LIN {X 0,Y 320.721,Z 461.024,A -85,B 0,C 180,E1 14265.571,E2 14265.571} C_VEL
LIN {X 0,Y 324.146,Z 440.908,A -85,B 0,C 180,E1 14264.497,E2 14264.497} C_VEL
LIN {X 0,Y 326.822,Z 419.622,A -85,B 0,C 180,E1 14263.687,E2 14263.687} C_VEL
LIN {X 0,Y 328.726,Z 391.924,A -85,B 0,C 180,E1 14262.985,E2 14262.985} C_VEL
LIN {X 0,Y 338,Z 225.821,A -85,B 0,C 180,E1 14259.275,E2 14259.275} C_VEL
LIN {X 0,Y 329.045,Z 209.572,A -85,B 0,C 180,E1 14256.958,E2 14256.958} C_VEL
LIN {X 0,Y 319.904,Z 194.705,A -85,B 0,C 180,E1 14254.397,E2 14254.397} C_VEL
LIN {X 0,Y 311.751,Z 182.649,A -85,B 0,C 180,E1 14251.896,E2 14251.896} C_VEL
LIN {X 0,Y 304.402,Z 172.591,A -85,B 0,C 180,E1 14249.41,E2 14249.41} C_VEL
LIN {X 0,Y 300.146,Z 166.89,A -85,B 0,C 180,E1 14247.799,E2 14247.799} C_VEL
LIN {X 0,Y 298.243,Z 163.151,A -85,B 0,C 180,E1 14246.265,E2 14246.265} C_VEL
LIN {X 0,Y 296.215,Z 159.192,A -85,B 0,C 180,E1 14244.53,E2 14244.53} C_VEL
LIN {X 0,Y 293.902,Z 154.755,A -85,B 0,C 180,E1 14242.397,E2 14242.397} C_VEL
LIN {X 0,Y 291.414,Z 150.066,A -85,B 0,C 180,E1 14239.857,E2 14239.857} C_VEL
LIN {X 0,Y 289.224,Z 146.434,A -85,B 0,C 180,E1 14237.503,E2 14237.503} C_VEL
LIN {X 0,Y 288.678,Z 145.099,A -85,B 0,C 180,E1 14236.707,E2 14236.707} C_VEL
LIN {X 0,Y 286.248,Z 141.602,A -85,B 0,C 180,E1 14233.74,E2 14233.74} C_VEL
LIN {X 0,Y 285.546,Z 139.698,A -85,B 0,C 180,E1 14232.333,E2 14232.333} C_VEL
LIN {X 0,Y 282.546,Z 135.185,A -85,B 0,C 180,E1 14226.706,E2 14226.706} C_VEL
LIN {X 0,Y 282.361,Z 134.287,A -85,B 0,C 180,E1 14225.282,E2 14225.282} C_VEL
LIN {X 0,Y 282.385,Z 134.265,A -85,B 0,C 180,E1 14220.608,E2 14220.608} C_VEL
LIN {X 0,Y 282.364,Z 134.277,A -85,B 0,C 180,E1 14215.938,E2 14215.938} C_VEL
LIN {X 0,Y 282.367,Z 134.308,A -85,B 0,C 180,E1 14211.08,E2 14211.08} C_VEL
LIN {X 0,Y 282.386,Z 134.493,A -85,B 0,C 180,E1 14209.596,E2 14209.596} C_VEL
LIN {X 0,Y 285.488,Z 139.677,A -85,B 0,C 180,E1 14203.1,E2 14203.1} C_VEL
LIN {X 0,Y 287.933,Z 144.473,A -85,B 0,C 180,E1 14199.255,E2 14199.255} C_VEL
LIN {X 0,Y 288.686,Z 145.379,A -85,B 0,C 180,E1 14198.461,E2 14198.461} C_VEL
LIN {X 0,Y 290.754,Z 149.516,A -85,B 0,C 180,E1 14195.843,E2 14195.843} C_VEL
LIN {X 0,Y 291.496,Z 150.817,A -85,B 0,C 180,E1 14195.045,E2 14195.045} C_VEL
LIN {X 0,Y 293.977,Z 155.554,A -85,B 0,C 180,E1 14192.447,E2 14192.447} C_VEL
LIN {X 0,Y 296.448,Z 160.545,A -85,B 0,C 180,E1 14190.054,E2 14190.054} C_VEL
LIN {X 0,Y 298.913,Z 165.761,A -85,B 0,C 180,E1 14187.807,E2 14187.807} C_VEL
LIN {X 0,Y 301.789,Z 171.506,A -85,B 0,C 180,E1 14185.605,E2 14185.605} C_VEL
LIN {X 0,Y 311.109,Z 184.598,A -85,B 0,C 180,E1 14182.393,E2 14182.393} C_VEL
LIN {X 0,Y 320.388,Z 199.042,A -85,B 0,C 180,E1 14179.556,E2 14179.556} C_VEL
LIN {X 0,Y 328.765,Z 213.325,A -85,B 0,C 180,E1 14177.237,E2 14177.237} C_VEL
LIN {X 0,Y 336.573,Z 228.034,A -85,B 0,C 180,E1 14175.231,E2 14175.231} C_VEL
LIN {X 0,Y 328.531,Z 396.994,A -85,B 0,C 180,E1 14171.76,E2 14171.76} C_VEL
LIN {X 0,Y 326.621,Z 416.539,A -85,B 0,C 180,E1 14171.071,E2 14171.071} C_VEL
LIN {X 0,Y 323.946,Z 435.192,A -85,B 0,C 180,E1 14170.112,E2 14170.112} C_VEL
LIN {X 0,Y 320.478,Z 453.585,A -85,B 0,C 180,E1 14168.835,E2 14168.835} C_VEL
LIN {X 0,Y 316.353,Z 471.266,A -85,B 0,C 180,E1 14167.245,E2 14167.245} C_VEL
LIN {X 0,Y 311.828,Z 487.803,A -85,B 0,C 180,E1 14165.362,E2 14165.362} C_VEL
LIN {X 0,Y 307.028,Z 503.233,A -85,B 0,C 180,E1 14163.167,E2 14163.167} C_VEL
LIN {X 0,Y 302.064,Z 517.674,A -85,B 0,C 180,E1 14160.612,E2 14160.612} C_VEL
LIN {X 0,Y 297.429,Z 530.269,A -85,B 0,C 180,E1 14157.856,E2 14157.856} C_VEL
LIN {X 0,Y 293.106,Z 541.516,A -85,B 0,C 180,E1 14154.807,E2 14154.807} C_VEL
LIN {X 0,Y 289.281,Z 551.303,A -85,B 0,C 180,E1 14151.491,E2 14151.491} C_VEL
LIN {X 0,Y 286.105,Z 559.611,A -85,B 0,C 180,E1 14147.909,E2 14147.909} C_VEL
LIN {X 0,Y 283.655,Z 566.396,A -85,B 0,C 180,E1 14144.075,E2 14144.075} C_VEL
LIN {X 0,Y 281.992,Z 571.558,A -85,B 0,C 180,E1 14140.004,E2 14140.004} C_VEL
LIN {X 0,Y 281.088,Z 574.878,A -85,B 0,C 180,E1 14135.92,E2 14135.92} C_VEL
LIN {X 0,Y 280.737,Z 576.48,A -85,B 0,C 180,E1 14131.836,E2 14131.836} C_VEL
LIN {X 0,Y 280.743,Z 576.471,A -85,B 0,C 180,E1 14127.958,E2 14127.958} C_VEL
LIN {X 0,Y 281.107,Z 574.834,A -85,B 0,C 180,E1 14123.873,E2 14123.873} C_VEL
LIN {X 0,Y 282.033,Z 571.47,A -85,B 0,C 180,E1 14119.789,E2 14119.789} C_VEL
LIN {X 0,Y 283.72,Z 566.25,A -85,B 0,C 180,E1 14115.717,E2 14115.717} C_VEL
LIN {X 0,Y 286.247,Z 559.287,A -85,B 0,C 180,E1 14111.824,E2 14111.824} C_VEL
LIN {X 0,Y 289.412,Z 551.061,A -85,B 0,C 180,E1 14108.304,E2 14108.304} C_VEL
LIN {X 0,Y 293.265,Z 541.222,A -85,B 0,C 180,E1 14104.989,E2 14104.989} C_VEL
LIN {X 0,Y 297.622,Z 529.918,A -85,B 0,C 180,E1 14101.943,E2 14101.943} C_VEL
LIN {X 0,Y 302.334,Z 517.118,A -85,B 0,C 180,E1 14099.161,E2 14099.161} C_VEL
LIN {X 0,Y 307.275,Z 502.717,A -85,B 0,C 180,E1 14096.637,E2 14096.637} C_VEL
LIN {X 0,Y 311.997,Z 487.513,A -85,B 0,C 180,E1 14094.489,E2 14094.489} C_VEL
LIN {X 0,Y 316.644,Z 470.484,A -85,B 0,C 180,E1 14092.564,E2 14092.564} C_VEL
LIN {X 0,Y 320.779,Z 452.575,A -85,B 0,C 180,E1 14090.976,E2 14090.976} C_VEL
LIN {X 0,Y 324.146,Z 434.561,A -85,B 0,C 180,E1 14089.741,E2 14089.741} C_VEL
LIN {X 0,Y 326.883,Z 415.161,A -85,B 0,C 180,E1 14088.763,E2 14088.763} C_VEL
LIN {X 0,Y 328.72,Z 395.639,A -85,B 0,C 180,E1 14088.095,E2 14088.095} C_VEL
LIN {X 0,Y 328.948,Z 391.546,A -85,B 0,C 180,E1 14087.996,E2 14087.996} C_VEL
LIN {X 0,Y 328.662,Z 383.97,A -85,B 0,C 180,E1 14087.703,E2 14087.703} C_VEL
LIN {X 0,Y 325.178,Z 364.134,A -85,B 0,C 180,E1 14086.515,E2 14086.515} C_VEL
LIN {X 0,Y 324.95,Z 357.606,A -85,B 0,C 180,E1 14086.286,E2 14086.286} C_VEL
LIN {X 0,Y 331.098,Z 230.961,A -85,B 0,C 180,E1 14083.663,E2 14083.663} C_VEL
LIN {X 0,Y 327.126,Z 223.644,A -85,B 0,C 180,E1 14082.619,E2 14082.619} C_VEL
LIN {X 0,Y 322.19,Z 240.736,A -85,B 0,C 180,E1 14082.119,E2 14082.119} C_VEL
LIN {X 0,Y 318.657,Z 249.667,A -85,B 0,C 180,E1 14081.638,E2 14081.638} C_VEL
LIN {X 0,Y 315.945,Z 253.882,A -85,B 0,C 180,E1 14081.167,E2 14081.167} C_VEL
LIN {X 0,Y 310.096,Z 277.776,A -85,B 0,C 180,E1 14080.634,E2 14080.634} C_VEL
LIN {X 0,Y 305.852,Z 291.273,A -85,B 0,C 180,E1 14080.092,E2 14080.092} C_VEL
LIN {X 0,Y 303.317,Z 296.772,A -85,B 0,C 180,E1 14079.663,E2 14079.663} C_VEL
LIN {X 0,Y 302.255,Z 297.734,A -85,B 0,C 180,E1 14079.431,E2 14079.431} C_VEL
LIN {X 0,Y 301.562,Z 297.398,A -85,B 0,C 180,E1 14079.232,E2 14079.232} C_VEL
LIN {X 0,Y 294.369,Z 406.379,A -85,B 0,C 180,E1 14075.561,E2 14075.561} C_VEL
LIN {X 0,Y 292.736,Z 426.04,A -85,B 0,C 180,E1 14074.541,E2 14074.541} C_VEL
LIN {X 0,Y 290.634,Z 445.674,A -85,B 0,C 180,E1 14073.162,E2 14073.162} C_VEL
LIN {X 0,Y 288.148,Z 465.179,A -85,B 0,C 180,E1 14071.392,E2 14071.392} C_VEL
LIN {X 0,Y 285.509,Z 483.447,A -85,B 0,C 180,E1 14069.306,E2 14069.306} C_VEL
LIN {X 0,Y 282.826,Z 500.339,A -85,B 0,C 180,E1 14066.905,E2 14066.905} C_VEL
LIN {X 0,Y 280.181,Z 516.365,A -85,B 0,C 180,E1 14064.118,E2 14064.118} C_VEL
LIN {X 0,Y 277.986,Z 529.646,A -85,B 0,C 180,E1 14061.302,E2 14061.302} C_VEL
LIN {X 0,Y 276.057,Z 541.908,A -85,B 0,C 180,E1 14058.149,E2 14058.149} C_VEL
LIN {X 0,Y 274.546,Z 552.542,A -85,B 0,C 180,E1 14054.77,E2 14054.77} C_VEL
LIN {X 0,Y 273.541,Z 561.1,A -85,B 0,C 180,E1 14051.384,E2 14051.384} C_VEL
LIN {X 0,Y 272.959,Z 567.848,A -85,B 0,C 180,E1 14048.002,E2 14048.002} C_VEL
LIN {X 0,Y 272.693,Z 573.226,A -85,B 0,C 180,E1 14044.417,E2 14044.417} C_VEL
LIN {X 0,Y 272.715,Z 576.877,A -85,B 0,C 180,E1 14040.841,E2 14040.841} C_VEL
LIN {X 0,Y 272.972,Z 578.945,A -85,B 0,C 180,E1 14037.271,E2 14037.271} C_VEL
LIN {X 0,Y 273.575,Z 579.472,A -85,B 0,C 180,E1 14033.706,E2 14033.706} C_VEL
LIN {X 0,Y 274.739,Z 578.347,A -85,B 0,C 180,E1 14029.94,E2 14029.94} C_VEL
LIN {X 0,Y 276.715,Z 575.316,A -85,B 0,C 180,E1 14025.99,E2 14025.99} C_VEL
LIN {X 0,Y 279.429,Z 570.626,A -85,B 0,C 180,E1 14022.293,E2 14022.293} C_VEL
LIN {X 0,Y 283.051,Z 564.115,A -85,B 0,C 180,E1 14018.664,E2 14018.664} C_VEL
LIN {X 0,Y 287.63,Z 555.651,A -85,B 0,C 180,E1 14015.127,E2 14015.127} C_VEL
LIN {X 0,Y 293.172,Z 544.938,A -85,B 0,C 180,E1 14011.702,E2 14011.702} C_VEL
LIN {X 0,Y 299.352,Z 532.673,A -85,B 0,C 180,E1 14008.598,E2 14008.598} C_VEL
LIN {X 0,Y 306.045,Z 518.945,A -85,B 0,C 180,E1 14005.811,E2 14005.811} C_VEL
LIN {X 0,Y 313.592,Z 502.655,A -85,B 0,C 180,E1 14003.172,E2 14003.172} C_VEL
LIN {X 0,Y 321.286,Z 485.354,A -85,B 0,C 180,E1 14000.936,E2 14000.936} C_VEL
LIN {X 0,Y 329.179,Z 466.218,A -85,B 0,C 180,E1 13998.999,E2 13998.999} C_VEL
LIN {X 0,Y 334.923,Z 451.016,A -85,B 0,C 180,E1 13997.764,E2 13997.764} C_VEL
LIN {X 0,Y 327.883,Z 467.006,A -85,B 0,C 180,E1 13996.661,E2 13996.661} C_VEL
LIN {X 0,Y 317.774,Z 488.595,A -85,B 0,C 180,E1 13994.688,E2 13994.688} C_VEL
LIN {X 0,Y 307.136,Z 511.532,A -85,B 0,C 180,E1 13991.865,E2 13991.865} C_VEL
LIN {X 0,Y 299.2,Z 529.521,A -85,B 0,C 180,E1 13989.046,E2 13989.046} C_VEL
LIN {X 0,Y 292.408,Z 545.751,A -85,B 0,C 180,E1 13986.026,E2 13986.026} C_VEL
LIN {X 0,Y 284.196,Z 568.647,A -85,B 0,C 180,E1 13980.859,E2 13980.859} C_VEL
LIN {X 0,Y 280.048,Z 581.452,A -85,B 0,C 180,E1 13977.252,E2 13977.252} C_VEL
LIN {X 0,Y 276.758,Z 592.506,A -85,B 0,C 180,E1 13973.417,E2 13973.417} C_VEL
LIN {X 0,Y 274.48,Z 601.426,A -85,B 0,C 180,E1 13969.582,E2 13969.582} C_VEL
LIN {X 0,Y 273.025,Z 608.934,A -85,B 0,C 180,E1 13965.507,E2 13965.507} C_VEL
LIN {X 0,Y 272.375,Z 614.641,A -85,B 0,C 180,E1 13961.435,E2 13961.435} C_VEL
LIN {X 0,Y 272.292,Z 618.543,A -85,B 0,C 180,E1 13957.385,E2 13957.385} C_VEL
LIN {X 0,Y 272.44,Z 620.7,A -85,B 0,C 180,E1 13953.578,E2 13953.578} C_VEL
LIN {X 0,Y 272.538,Z 621.429,A -85,B 0,C 180,E1 13950.001,E2 13950.001} C_VEL
LIN {X 0,Y 272.44,Z 620.694,A -85,B 0,C 180,E1 13946.424,E2 13946.424} C_VEL
LIN {X 0,Y 272.293,Z 618.427,A -85,B 0,C 180,E1 13942.494,E2 13942.494} C_VEL
LIN {X 0,Y 272.379,Z 614.605,A -85,B 0,C 180,E1 13938.553,E2 13938.553} C_VEL
LIN {X 0,Y 273.08,Z 608.583,A -85,B 0,C 180,E1 13934.281,E2 13934.281} C_VEL
LIN {X 0,Y 274.579,Z 600.957,A -85,B 0,C 180,E1 13930.207,E2 13930.207} C_VEL
LIN {X 0,Y 276.908,Z 591.911,A -85,B 0,C 180,E1 13926.373,E2 13926.373} C_VEL
LIN {X 0,Y 280.199,Z 580.888,A -85,B 0,C 180,E1 13922.594,E2 13922.594} C_VEL
LIN {X 0,Y 284.242,Z 568.375,A -85,B 0,C 180,E1 13919.099,E2 13919.099} C_VEL
LIN {X 0,Y 288.904,Z 554.372,A -85,B 0,C 180,E1 13915.9,E2 13915.9} C_VEL
LIN {X 0,Y 293.821,Z 539.443,A -85,B 0,C 180,E1 13913.1,E2 13913.1} C_VEL
LIN {X 0,Y 298.836,Z 523.569,A -85,B 0,C 180,E1 13910.653,E2 13910.653} C_VEL
LIN {X 0,Y 303.926,Z 506.248,A -85,B 0,C 180,E1 13908.481,E2 13908.481} C_VEL
LIN {X 0,Y 308.921,Z 487.336,A -85,B 0,C 180,E1 13906.585,E2 13906.585} C_VEL
LIN {X 0,Y 313.413,Z 467.675,A -85,B 0,C 180,E1 13905.04,E2 13905.04} C_VEL
LIN {X 0,Y 317.16,Z 447.865,A -85,B 0,C 180,E1 13903.853,E2 13903.853} C_VEL
LIN {X 0,Y 320.173,Z 427.576,A -85,B 0,C 180,E1 13902.971,E2 13902.971} C_VEL
LIN {X 0,Y 322.146,Z 406.936,A -85,B 0,C 180,E1 13902.343,E2 13902.343} C_VEL
LIN {X 0,Y 332.51,Z 229.162,A -85,B 0,C 180,E1 13898.33,E2 13898.33} C_VEL
LIN {X 0,Y 324.025,Z 213.704,A -85,B 0,C 180,E1 13896.03,E2 13896.03} C_VEL
LIN {X 0,Y 315.35,Z 199.501,A -85,B 0,C 180,E1 13893.483,E2 13893.483} C_VEL
LIN {X 0,Y 308.132,Z 188.679,A -85,B 0,C 180,E1 13891.168,E2 13891.168} C_VEL
LIN {X 0,Y 301.292,Z 179.158,A -85,B 0,C 180,E1 13888.763,E2 13888.763} C_VEL
LIN {X 0,Y 294.67,Z 170.446,A -85,B 0,C 180,E1 13886.174,E2 13886.174} C_VEL
LIN {X 0,Y 292.225,Z 167.155,A -85,B 0,C 180,E1 13885.104,E2 13885.104} C_VEL
LIN {X 0,Y 289.065,Z 161.017,A -85,B 0,C 180,E1 13882.149,E2 13882.149} C_VEL
LIN {X 0,Y 286.6,Z 156.365,A -85,B 0,C 180,E1 13879.567,E2 13879.567} C_VEL
LIN {X 0,Y 284.396,Z 152.307,A -85,B 0,C 180,E1 13876.966,E2 13876.966} C_VEL
LIN {X 0,Y 281.446,Z 147.281,A -85,B 0,C 180,E1 13872.933,E2 13872.933} C_VEL
LIN {X 0,Y 281.023,Z 146.284,A -85,B 0,C 180,E1 13872.117,E2 13872.117} C_VEL
LIN {X 0,Y 278.061,Z 141.193,A -85,B 0,C 180,E1 13865.778,E2 13865.778} C_VEL
LIN {X 0,Y 276.494,Z 139.699,A -85,B 0,C 180,E1 13860,E2 13860} C_VEL
LIN {X 0,Y 276.627,Z 139.823,A -85,B 0,C 180,E1 13854.399,E2 13854.399} C_VEL
LIN {X 0,Y 278.003,Z 141.235,A -85,B 0,C 180,E1 13849.64,E2 13849.64} C_VEL
LIN {X 0,Y 281.141,Z 146.703,A -85,B 0,C 180,E1 13842.831,E2 13842.831} C_VEL
LIN {X 0,Y 283.149,Z 150.815,A -85,B 0,C 180,E1 13839.537,E2 13839.537} C_VEL
LIN {X 0,Y 283.991,Z 152.057,A -85,B 0,C 180,E1 13838.521,E2 13838.521} C_VEL
LIN {X 0,Y 286.629,Z 157.135,A -85,B 0,C 180,E1 13835.253,E2 13835.253} C_VEL
LIN {X 0,Y 289.044,Z 161.888,A -85,B 0,C 180,E1 13832.608,E2 13832.608} C_VEL
LIN {X 0,Y 291.452,Z 166.908,A -85,B 0,C 180,E1 13830.169,E2 13830.169} C_VEL
LIN {X 0,Y 293.543,Z 171.094,A -85,B 0,C 180,E1 13828.361,E2 13828.361} C_VEL
LIN {X 0,Y 300.954,Z 181.269,A -85,B 0,C 180,E1 13825.439,E2 13825.439} C_VEL
LIN {X 0,Y 308.11,Z 191.569,A -85,B 0,C 180,E1 13822.93,E2 13822.93} C_VEL
LIN {X 0,Y 316.276,Z 204.433,A -85,B 0,C 180,E1 13820.342,E2 13820.342} C_VEL
LIN {X 0,Y 324.485,Z 218.621,A -85,B 0,C 180,E1 13817.976,E2 13817.976} C_VEL
LIN {X 0,Y 331.104,Z 231.411,A -85,B 0,C 180,E1 13816.191,E2 13816.191} C_VEL
LIN {X 0,Y 322.837,Z 397.249,A -85,B 0,C 180,E1 13812.748,E2 13812.748} C_VEL
LIN {X 0,Y 320.848,Z 416.862,A -85,B 0,C 180,E1 13812.051,E2 13812.051} C_VEL
LIN {X 0,Y 318.044,Z 435.683,A -85,B 0,C 180,E1 13811.073,E2 13811.073} C_VEL
LIN {X 0,Y 314.5,Z 453.819,A -85,B 0,C 180,E1 13809.804,E2 13809.804} C_VEL
LIN {X 0,Y 310.283,Z 471.324,A -85,B 0,C 180,E1 13808.22,E2 13808.22} C_VEL
LIN {X 0,Y 305.572,Z 487.939,A -85,B 0,C 180,E1 13806.315,E2 13806.315} C_VEL
LIN {X 0,Y 300.485,Z 503.681,A -85,B 0,C 180,E1 13804.05,E2 13804.05} C_VEL
LIN {X 0,Y 295.609,Z 517.34,A -85,B 0,C 180,E1 13801.617,E2 13801.617} C_VEL
LIN {X 0,Y 290.678,Z 530.198,A -85,B 0,C 180,E1 13798.786,E2 13798.786} C_VEL
LIN {X 0,Y 285.946,Z 541.951,A -85,B 0,C 180,E1 13795.558,E2 13795.558} C_VEL
LIN {X 0,Y 281.828,Z 551.972,A -85,B 0,C 180,E1 13792.088,E2 13792.088} C_VEL
LIN {X 0,Y 278.476,Z 560.272,A -85,B 0,C 180,E1 13788.417,E2 13788.417} C_VEL
LIN {X 0,Y 275.88,Z 567.05,A -85,B 0,C 180,E1 13784.48,E2 13784.48} C_VEL
LIN {X 0,Y 274.109,Z 572.208,A -85,B 0,C 180,E1 13780.295,E2 13780.295} C_VEL
LIN {X 0,Y 273.141,Z 575.525,A -85,B 0,C 180,E1 13776.092,E2 13776.092} C_VEL
LIN {X 0,Y 272.766,Z 577.125,A -85,B 0,C 180,E1 13771.889,E2 13771.889} C_VEL
LIN {X 0,Y 272.772,Z 577.116,A -85,B 0,C 180,E1 13767.898,E2 13767.898} C_VEL
LIN {X 0,Y 273.162,Z 575.48,A -85,B 0,C 180,E1 13763.694,E2 13763.694} C_VEL
LIN {X 0,Y 274.153,Z 572.119,A -85,B 0,C 180,E1 13759.492,E2 13759.492} C_VEL
LIN {X 0,Y 275.95,Z 566.904,A -85,B 0,C 180,E1 13755.306,E2 13755.306} C_VEL
LIN {X 0,Y 278.597,Z 560.031,A -85,B 0,C 180,E1 13751.348,E2 13751.348} C_VEL
LIN {X 0,Y 281.967,Z 551.729,A -85,B 0,C 180,E1 13747.701,E2 13747.701} C_VEL
LIN {X 0,Y 286.015,Z 541.9,A -85,B 0,C 180,E1 13744.31,E2 13744.31} C_VEL
LIN {X 0,Y 290.575,Z 530.609,A -85,B 0,C 180,E1 13741.2,E2 13741.2} C_VEL
LIN {X 0,Y 295.493,Z 517.829,A -85,B 0,C 180,E1 13738.366,E2 13738.366} C_VEL
LIN {X 0,Y 300.638,Z 503.463,A -85,B 0,C 180,E1 13735.801,E2 13735.801} C_VEL
LIN {X 0,Y 305.596,Z 488.133,A -85,B 0,C 180,E1 13733.599,E2 13733.599} C_VEL
LIN {X 0,Y 310.331,Z 471.48,A -85,B 0,C 180,E1 13731.685,E2 13731.685} C_VEL
LIN {X 0,Y 314.652,Z 453.578,A -85,B 0,C 180,E1 13730.066,E2 13730.066} C_VEL
LIN {X 0,Y 318.258,Z 435.042,A -85,B 0,C 180,E1 13728.778,E2 13728.778} C_VEL
LIN {X 0,Y 321.1,Z 415.675,A -85,B 0,C 180,E1 13727.789,E2 13727.789} C_VEL
LIN {X 0,Y 323.029,Z 395.937,A -85,B 0,C 180,E1 13727.107,E2 13727.107} C_VEL
LIN {X 0,Y 324.95,Z 357.606,A -85,B 0,C 180,E1 13726.286,E2 13726.286} C_VEL
LIN {X 0,Y 324.621,Z 350.016,A -85,B 0,C 180,E1 13726.001,E2 13726.001} C_VEL
LIN {X 0,Y 321.36,Z 330.183,A -85,B 0,C 180,E1 13724.779,E2 13724.779} C_VEL
LIN {X 0,Y 321.186,Z 323.658,A -85,B 0,C 180,E1 13724.544,E2 13724.544} C_VEL
LIN {X 0,Y 325.081,Z 248.133,A -85,B 0,C 180,E1 13722.974,E2 13722.974} C_VEL
LIN {X 0,Y 321.526,Z 255.837,A -85,B 0,C 180,E1 13722.47,E2 13722.47} C_VEL
LIN {X 0,Y 319.946,Z 258.655,A -85,B 0,C 180,E1 13722.221,E2 13722.221} C_VEL
LIN {X 0,Y 314.67,Z 280.015,A -85,B 0,C 180,E1 13721.766,E2 13721.766} C_VEL
LIN {X 0,Y 310.18,Z 294.181,A -85,B 0,C 180,E1 13721.224,E2 13721.224} C_VEL
LIN {X 0,Y 307.045,Z 301.133,A -85,B 0,C 180,E1 13720.731,E2 13720.731} C_VEL
LIN {X 0,Y 305.019,Z 304.248,A -85,B 0,C 180,E1 13720.355,E2 13720.355} C_VEL
LIN {X 0,Y 299.822,Z 325.845,A -85,B 0,C 180,E1 13719.853,E2 13719.853} C_VEL
LIN {X 0,Y 295.477,Z 340.074,A -85,B 0,C 180,E1 13719.272,E2 13719.272} C_VEL
LIN {X 0,Y 292.906,Z 345.871,A -85,B 0,C 180,E1 13718.816,E2 13718.816} C_VEL
LIN {X 0,Y 291.843,Z 347.012,A -85,B 0,C 180,E1 13718.575,E2 13718.575} C_VEL
LIN {X 0,Y 291.014,Z 346.438,A -85,B 0,C 180,E1 13718.328,E2 13718.328} C_VEL
LIN {X 0,Y 286.914,Z 407.955,A -85,B 0,C 180,E1 13716.121,E2 13716.121} C_VEL
LIN {X 0,Y 285.095,Z 428.59,A -85,B 0,C 180,E1 13714.989,E2 13714.989} C_VEL
LIN {X 0,Y 282.789,Z 448.937,A -85,B 0,C 180,E1 13713.475,E2 13713.475} C_VEL
LIN {X 0,Y 280.212,Z 468.091,A -85,B 0,C 180,E1 13711.637,E2 13711.637} C_VEL
LIN {X 0,Y 277.478,Z 486.024,A -85,B 0,C 180,E1 13709.464,E2 13709.464} C_VEL
LIN {X 0,Y 274.813,Z 502.251,A -85,B 0,C 180,E1 13707.052,E2 13707.052} C_VEL
LIN {X 0,Y 272.218,Z 517.527,A -85,B 0,C 180,E1 13704.292,E2 13704.292} C_VEL
LIN {X 0,Y 269.902,Z 531.224,A -85,B 0,C 180,E1 13701.288,E2 13701.288} C_VEL
LIN {X 0,Y 267.958,Z 543.317,A -85,B 0,C 180,E1 13698.042,E2 13698.042} C_VEL
LIN {X 0,Y 266.454,Z 553.846,A -85,B 0,C 180,E1 13694.562,E2 13694.562} C_VEL
LIN {X 0,Y 265.472,Z 562.329,A -85,B 0,C 180,E1 13691.075,E2 13691.075} C_VEL
LIN {X 0,Y 264.89,Z 569.318,A -85,B 0,C 180,E1 13687.374,E2 13687.374} C_VEL
LIN {X 0,Y 264.685,Z 574.489,A -85,B 0,C 180,E1 13683.682,E2 13683.682} C_VEL
LIN {X 0,Y 264.767,Z 577.987,A -85,B 0,C 180,E1 13680,E2 13680} C_VEL
LIN {X 0,Y 265.119,Z 579.888,A -85,B 0,C 180,E1 13676.325,E2 13676.325} C_VEL
LIN {X 0,Y 265.936,Z 580.237,A -85,B 0,C 180,E1 13672.439,E2 13672.439} C_VEL
LIN {X 0,Y 267.384,Z 578.896,A -85,B 0,C 180,E1 13668.569,E2 13668.569} C_VEL
LIN {X 0,Y 269.768,Z 575.645,A -85,B 0,C 180,E1 13664.523,E2 13664.523} C_VEL
LIN {X 0,Y 272.954,Z 570.781,A -85,B 0,C 180,E1 13660.751,E2 13660.751} C_VEL
LIN {X 0,Y 277.103,Z 564.084,A -85,B 0,C 180,E1 13657.065,E2 13657.065} C_VEL
LIN {X 0,Y 282.255,Z 555.427,A -85,B 0,C 180,E1 13653.491,E2 13653.491} C_VEL
LIN {X 0,Y 288.45,Z 544.687,A -85,B 0,C 180,E1 13650.057,E2 13650.057} C_VEL
LIN {X 0,Y 295.292,Z 532.463,A -85,B 0,C 180,E1 13646.966,E2 13646.966} C_VEL
LIN {X 0,Y 303.102,Z 517.88,A -85,B 0,C 180,E1 13644.043,E2 13644.043} C_VEL
LIN {X 0,Y 311.438,Z 501.826,A -85,B 0,C 180,E1 13641.477,E2 13641.477} C_VEL
LIN {X 0,Y 320.133,Z 484.088,A -85,B 0,C 180,E1 13639.25,E2 13639.25} C_VEL
LIN {X 0,Y 326.254,Z 470.856,A -85,B 0,C 180,E1 13637.873,E2 13637.873} C_VEL
LIN {X 0,Y 315.193,Z 491.782,A -85,B 0,C 180,E1 13635.932,E2 13635.932} C_VEL
LIN {X 0,Y 303.727,Z 513.213,A -85,B 0,C 180,E1 13633.216,E2 13633.216} C_VEL
LIN {X 0,Y 295.284,Z 529.771,A -85,B 0,C 180,E1 13630.553,E2 13630.553} C_VEL
LIN {X 0,Y 287.13,Z 546.646,A -85,B 0,C 180,E1 13627.296,E2 13627.296} C_VEL
LIN {X 0,Y 279.86,Z 563.286,A -85,B 0,C 180,E1 13623.382,E2 13623.382} C_VEL
LIN {X 0,Y 274.124,Z 577.633,A -85,B 0,C 180,E1 13619.26,E2 13619.26} C_VEL
LIN {X 0,Y 269.875,Z 589.787,A -85,B 0,C 180,E1 13614.985,E2 13614.985} C_VEL
LIN {X 0,Y 266.841,Z 600.351,A -85,B 0,C 180,E1 13610.395,E2 13610.395} C_VEL
LIN {X 0,Y 265.118,Z 608.397,A -85,B 0,C 180,E1 13605.91,E2 13605.91} C_VEL
LIN {X 0,Y 264.389,Z 614.215,A -85,B 0,C 180,E1 13601.564,E2 13601.564} C_VEL
LIN {X 0,Y 264.303,Z 617.89,A -85,B 0,C 180,E1 13597.61,E2 13597.61} C_VEL
LIN {X 0,Y 264.457,Z 620.053,A -85,B 0,C 180,E1 13593.687,E2 13593.687} C_VEL
LIN {X 0,Y 264.564,Z 620.784,A -85,B 0,C 180,E1 13590.001,E2 13590.001} C_VEL
LIN {X 0,Y 264.457,Z 620.046,A -85,B 0,C 180,E1 13586.316,E2 13586.316} C_VEL
LIN {X 0,Y 264.304,Z 617.853,A -85,B 0,C 180,E1 13582.366,E2 13582.366} C_VEL
LIN {X 0,Y 264.41,Z 613.961,A -85,B 0,C 180,E1 13578.219,E2 13578.219} C_VEL
LIN {X 0,Y 265.199,Z 607.913,A -85,B 0,C 180,E1 13573.801,E2 13573.801} C_VEL
LIN {X 0,Y 266.837,Z 600.276,A -85,B 0,C 180,E1 13569.607,E2 13569.607} C_VEL
LIN {X 0,Y 269.346,Z 591.217,A -85,B 0,C 180,E1 13565.668,E2 13565.668} C_VEL
LIN {X 0,Y 272.872,Z 580.18,A -85,B 0,C 180,E1 13561.793,E2 13561.793} C_VEL
LIN {X 0,Y 277.169,Z 567.648,A -85,B 0,C 180,E1 13558.22,E2 13558.22} C_VEL
LIN {X 0,Y 282.093,Z 553.62,A -85,B 0,C 180,E1 13554.958,E2 13554.958} C_VEL
LIN {X 0,Y 287.285,Z 538.596,A -85,B 0,C 180,E1 13552.102,E2 13552.102} C_VEL
LIN {X 0,Y 292.498,Z 522.805,A -85,B 0,C 180,E1 13549.641,E2 13549.641} C_VEL
LIN {X 0,Y 297.826,Z 505.403,A -85,B 0,C 180,E1 13547.44,E2 13547.44} C_VEL
LIN {X 0,Y 302.862,Z 487.04,A -85,B 0,C 180,E1 13545.584,E2 13545.584} C_VEL
LIN {X 0,Y 307.439,Z 467.75,A -85,B 0,C 180,E1 13544.052,E2 13544.052} C_VEL
LIN {X 0,Y 311.313,Z 448.08,A -85,B 0,C 180,E1 13542.857,E2 13542.857} C_VEL
LIN {X 0,Y 314.439,Z 427.882,A -85,B 0,C 180,E1 13541.965,E2 13541.965} C_VEL
LIN {X 0,Y 316.518,Z 407.161,A -85,B 0,C 180,E1 13541.323,E2 13541.323} C_VEL
LIN {X 0,Y 327.07,Z 232.467,A -85,B 0,C 180,E1 13537.344,E2 13537.344} C_VEL
LIN {X 0,Y 318.567,Z 216.918,A -85,B 0,C 180,E1 13534.918,E2 13534.918} C_VEL
LIN {X 0,Y 310.267,Z 203.237,A -85,B 0,C 180,E1 13532.34,E2 13532.34} C_VEL
LIN {X 0,Y 302.22,Z 191.277,A -85,B 0,C 180,E1 13529.589,E2 13529.589} C_VEL
LIN {X 0,Y 295.158,Z 181.432,A -85,B 0,C 180,E1 13526.887,E2 13526.887} C_VEL
LIN {X 0,Y 288.122,Z 172.385,A -85,B 0,C 180,E1 13523.846,E2 13523.846} C_VEL
LIN {X 0,Y 284.234,Z 167.276,A -85,B 0,C 180,E1 13521.893,E2 13521.893} C_VEL
LIN {X 0,Y 281.798,Z 162.655,A -85,B 0,C 180,E1 13519.267,E2 13519.267} C_VEL
LIN {X 0,Y 279.168,Z 157.811,A -85,B 0,C 180,E1 13516.008,E2 13516.008} C_VEL
LIN {X 0,Y 276.923,Z 153.822,A -85,B 0,C 180,E1 13512.723,E2 13512.723} C_VEL
LIN {X 0,Y 276.494,Z 152.864,A -85,B 0,C 180,E1 13511.895,E2 13511.895} C_VEL
LIN {X 0,Y 273.519,Z 147.617,A -85,B 0,C 180,E1 13505.033,E2 13505.033} C_VEL
LIN {X 0,Y 272.086,Z 146.325,A -85,B 0,C 180,E1 13498.526,E2 13498.526} C_VEL
LIN {X 0,Y 272.638,Z 146.904,A -85,B 0,C 180,E1 13492.837,E2 13492.837} C_VEL
LIN {X 0,Y 273.622,Z 147.974,A -85,B 0,C 180,E1 13489.685,E2 13489.685} C_VEL
LIN {X 0,Y 276.556,Z 153.306,A -85,B 0,C 180,E1 13482.971,E2 13482.971} C_VEL
LIN {X 0,Y 278.746,Z 157.548,A -85,B 0,C 180,E1 13479.419,E2 13479.419} C_VEL
LIN {X 0,Y 281.77,Z 163.445,A -85,B 0,C 180,E1 13475.469,E2 13475.469} C_VEL
LIN {X 0,Y 284.122,Z 168.211,A -85,B 0,C 180,E1 13472.775,E2 13472.775} C_VEL
LIN {X 0,Y 285.747,Z 171.162,A -85,B 0,C 180,E1 13471.355,E2 13471.355} C_VEL
LIN {X 0,Y 291.644,Z 179.101,A -85,B 0,C 180,E1 13468.65,E2 13468.65} C_VEL
LIN {X 0,Y 297.842,Z 187.7,A -85,B 0,C 180,E1 13466.133,E2 13466.133} C_VEL
LIN {X 0,Y 304.727,Z 197.796,A -85,B 0,C 180,E1 13463.624,E2 13463.624} C_VEL
LIN {X 0,Y 312.797,Z 210.774,A -85,B 0,C 180,E1 13460.971,E2 13460.971} C_VEL
LIN {X 0,Y 320.652,Z 224.68,A -85,B 0,C 180,E1 13458.619,E2 13458.619} C_VEL
LIN {X 0,Y 325.729,Z 234.726,A -85,B 0,C 180,E1 13457.186,E2 13457.186} C_VEL
LIN {X 0,Y 317.226,Z 397.666,A -85,B 0,C 180,E1 13453.766,E2 13453.766} C_VEL
LIN {X 0,Y 315.155,Z 417.294,A -85,B 0,C 180,E1 13453.061,E2 13453.061} C_VEL
LIN {X 0,Y 312.358,Z 435.507,A -85,B 0,C 180,E1 13452.112,E2 13452.112} C_VEL
LIN {X 0,Y 308.507,Z 454.52,A -85,B 0,C 180,E1 13450.77,E2 13450.77} C_VEL
LIN {X 0,Y 304.074,Z 472.189,A -85,B 0,C 180,E1 13449.147,E2 13449.147} C_VEL
LIN {X 0,Y 299.187,Z 488.734,A -85,B 0,C 180,E1 13447.219,E2 13447.219} C_VEL
LIN {X 0,Y 293.931,Z 504.349,A -85,B 0,C 180,E1 13444.934,E2 13444.934} C_VEL
LIN {X 0,Y 288.83,Z 518.062,A -85,B 0,C 180,E1 13442.449,E2 13442.449} C_VEL
LIN {X 0,Y 283.684,Z 530.897,A -85,B 0,C 180,E1 13439.565,E2 13439.565} C_VEL
LIN {X 0,Y 278.698,Z 542.703,A -85,B 0,C 180,E1 13436.245,E2 13436.245} C_VEL
LIN {X 0,Y 274.406,Z 552.639,A -85,B 0,C 180,E1 13432.719,E2 13432.719} C_VEL
LIN {X 0,Y 270.87,Z 560.932,A -85,B 0,C 180,E1 13428.954,E2 13428.954} C_VEL
LIN {X 0,Y 268.118,Z 567.704,A -85,B 0,C 180,E1 13424.909,E2 13424.909} C_VEL
LIN {X 0,Y 266.233,Z 572.857,A -85,B 0,C 180,E1 13420.603,E2 13420.603} C_VEL
LIN {X 0,Y 265.197,Z 576.171,A -85,B 0,C 180,E1 13416.276,E2 13416.276} C_VEL
LIN {X 0,Y 264.805,Z 577.74,A -85,B 0,C 180,E1 13412.163,E2 13412.163} C_VEL
LIN {X 0,Y 264.79,Z 577.782,A -85,B 0,C 180,E1 13408.051,E2 13408.051} C_VEL
LIN {X 0,Y 265.151,Z 576.335,A -85,B 0,C 180,E1 13403.938,E2 13403.938} C_VEL
LIN {X 0,Y 266.067,Z 573.344,A -85,B 0,C 180,E1 13399.826,E2 13399.826} C_VEL
LIN {X 0,Y 267.727,Z 568.708,A -85,B 0,C 180,E1 13395.729,E2 13395.729} C_VEL
LIN {X 0,Y 270.307,Z 562.287,A -85,B 0,C 180,E1 13391.673,E2 13391.673} C_VEL
LIN {X 0,Y 273.672,Z 554.369,A -85,B 0,C 180,E1 13387.893,E2 13387.893} C_VEL
LIN {X 0,Y 277.721,Z 545.014,A -85,B 0,C 180,E1 13384.402,E2 13384.402} C_VEL
LIN {X 0,Y 282.621,Z 533.523,A -85,B 0,C 180,E1 13381.007,E2 13381.007} C_VEL
LIN {X 0,Y 287.628,Z 521.227,A -85,B 0,C 180,E1 13378.102,E2 13378.102} C_VEL
LIN {X 0,Y 293.064,Z 506.904,A -85,B 0,C 180,E1 13375.384,E2 13375.384} C_VEL
LIN {X 0,Y 298.335,Z 491.588,A -85,B 0,C 180,E1 13373.057,E2 13373.057} C_VEL
LIN {X 0,Y 303.208,Z 475.517,A -85,B 0,C 180,E1 13371.1,E2 13371.1} C_VEL
LIN {X 0,Y 307.647,Z 458.513,A -85,B 0,C 180,E1 13369.457,E2 13369.457} C_VEL
LIN {X 0,Y 311.481,Z 440.656,A -85,B 0,C 180,E1 13368.11,E2 13368.11} C_VEL
LIN {X 0,Y 314.664,Z 421.436,A -85,B 0,C 180,E1 13367.023,E2 13367.023} C_VEL
LIN {X 0,Y 316.965,Z 401.616,A -85,B 0,C 180,E1 13366.247,E2 13366.247} C_VEL
LIN {X 0,Y 318.575,Z 375.681,A -85,B 0,C 180,E1 13365.624,E2 13365.624} C_VEL
LIN {X 0,Y 321.186,Z 323.658,A -85,B 0,C 180,E1 13364.544,E2 13364.544} C_VEL
LIN {X 0,Y 320.906,Z 316.068,A -85,B 0,C 180,E1 13364.254,E2 13364.254} C_VEL
LIN {X 0,Y 317.843,Z 296.246,A -85,B 0,C 180,E1 13362.994,E2 13362.994} C_VEL
LIN {X 0,Y 317.716,Z 289.721,A -85,B 0,C 180,E1 13362.755,E2 13362.755} C_VEL
LIN {X 0,Y 317.799,Z 287.595,A -85,B 0,C 180,E1 13362.704,E2 13362.704} C_VEL
LIN {X 0,Y 313.451,Z 300.051,A -85,B 0,C 180,E1 13362.165,E2 13362.165} C_VEL
LIN {X 0,Y 310.06,Z 306.801,A -85,B 0,C 180,E1 13361.629,E2 13361.629} C_VEL
LIN {X 0,Y 309.14,Z 308.553,A -85,B 0,C 180,E1 13361.478,E2 13361.478} C_VEL
LIN {X 0,Y 303.9,Z 329.612,A -85,B 0,C 180,E1 13360.985,E2 13360.985} C_VEL
LIN {X 0,Y 299.502,Z 343.572,A -85,B 0,C 180,E1 13360.422,E2 13360.422} C_VEL
LIN {X 0,Y 296.469,Z 350.354,A -85,B 0,C 180,E1 13359.914,E2 13359.914} C_VEL
LIN {X 0,Y 294.266,Z 353.664,A -85,B 0,C 180,E1 13359.473,E2 13359.473} C_VEL
LIN {X 0,Y 288.884,Z 375.988,A -85,B 0,C 180,E1 13358.909,E2 13358.909} C_VEL
LIN {X 0,Y 284.781,Z 389.185,A -85,B 0,C 180,E1 13358.31,E2 13358.31} C_VEL
LIN {X 0,Y 282.372,Z 393.868,A -85,B 0,C 180,E1 13357.857,E2 13357.857} C_VEL
LIN {X 0,Y 281.525,Z 394.662,A -85,B 0,C 180,E1 13357.653,E2 13357.653} C_VEL
LIN {X 0,Y 280.64,Z 394.231,A -85,B 0,C 180,E1 13357.374,E2 13357.374} C_VEL
LIN {X 0,Y 280.515,Z 394.039,A -85,B 0,C 180,E1 13357.321,E2 13357.321} C_VEL
LIN {X 0,Y 278.853,Z 416.391,A -85,B 0,C 180,E1 13356.329,E2 13356.329} C_VEL
LIN {X 0,Y 276.806,Z 436.465,A -85,B 0,C 180,E1 13355.053,E2 13355.053} C_VEL
LIN {X 0,Y 274.335,Z 456.227,A -85,B 0,C 180,E1 13353.391,E2 13353.391} C_VEL
LIN {X 0,Y 271.603,Z 475.04,A -85,B 0,C 180,E1 13351.381,E2 13351.381} C_VEL
LIN {X 0,Y 268.774,Z 492.588,A -85,B 0,C 180,E1 13349.045,E2 13349.045} C_VEL
LIN {X 0,Y 266.004,Z 508.643,A -85,B 0,C 180,E1 13346.411,E2 13346.411} C_VEL
LIN {X 0,Y 263.348,Z 523.818,A -85,B 0,C 180,E1 13343.376,E2 13343.376} C_VEL
LIN {X 0,Y 261.1,Z 537.004,A -85,B 0,C 180,E1 13340.161,E2 13340.161} C_VEL
LIN {X 0,Y 259.328,Z 548.237,A -85,B 0,C 180,E1 13336.809,E2 13336.809} C_VEL
LIN {X 0,Y 258.003,Z 557.962,A -85,B 0,C 180,E1 13333.218,E2 13333.218} C_VEL
LIN {X 0,Y 257.19,Z 565.734,A -85,B 0,C 180,E1 13329.624,E2 13329.624} C_VEL
LIN {X 0,Y 256.783,Z 571.787,A -85,B 0,C 180,E1 13326.035,E2 13326.035} C_VEL
LIN {X 0,Y 256.694,Z 576.474,A -85,B 0,C 180,E1 13322.233,E2 13322.233} C_VEL
LIN {X 0,Y 256.893,Z 579.516,A -85,B 0,C 180,E1 13318.439,E2 13318.439} C_VEL
LIN {X 0,Y 257.481,Z 581.04,A -85,B 0,C 180,E1 13314.429,E2 13314.429} C_VEL
LIN {X 0,Y 258.648,Z 580.869,A -85,B 0,C 180,E1 13310.432,E2 13310.432} C_VEL
LIN {X 0,Y 260.562,Z 579.025,A -85,B 0,C 180,E1 13306.463,E2 13306.463} C_VEL
LIN {X 0,Y 263.563,Z 575.26,A -85,B 0,C 180,E1 13302.333,E2 13302.333} C_VEL
LIN {X 0,Y 267.667,Z 569.592,A -85,B 0,C 180,E1 13298.297,E2 13298.297} C_VEL
LIN {X 0,Y 272.939,Z 561.933,A -85,B 0,C 180,E1 13294.389,E2 13294.389} C_VEL
LIN {X 0,Y 279.024,Z 552.656,A -85,B 0,C 180,E1 13290.834,E2 13290.834} C_VEL
LIN {X 0,Y 286.633,Z 540.633,A -85,B 0,C 180,E1 13287.27,E2 13287.27} C_VEL
LIN {X 0,Y 294.522,Z 527.799,A -85,B 0,C 180,E1 13284.274,E2 13284.274} C_VEL
LIN {X 0,Y 303.431,Z 512.656,A -85,B 0,C 180,E1 13281.48,E2 13281.48} C_VEL
LIN {X 0,Y 312.864,Z 496.081,A -85,B 0,C 180,E1 13279.07,E2 13279.07} C_VEL
LIN {X 0,Y 317.581,Z 487.365,A -85,B 0,C 180,E1 13277.99,E2 13277.99} C_VEL
LIN {X 0,Y 308.036,Z 503.062,A -85,B 0,C 180,E1 13276.239,E2 13276.239} C_VEL
LIN {X 0,Y 296.886,Z 521.583,A -85,B 0,C 180,E1 13273.608,E2 13273.608} C_VEL
LIN {X 0,Y 285.831,Z 541.017,A -85,B 0,C 180,E1 13270.066,E2 13270.066} C_VEL
LIN {X 0,Y 277.1,Z 557.578,A -85,B 0,C 180,E1 13266.283,E2 13266.283} C_VEL
LIN {X 0,Y 269.759,Z 572.916,A -85,B 0,C 180,E1 13262.009,E2 13262.009} C_VEL
LIN {X 0,Y 264.441,Z 585.47,A -85,B 0,C 180,E1 13257.716,E2 13257.716} C_VEL
LIN {X 0,Y 260.6,Z 595.993,A -85,B 0,C 180,E1 13253.279,E2 13253.279} C_VEL
LIN {X 0,Y 258.077,Z 604.479,A -85,B 0,C 180,E1 13248.759,E2 13248.759} C_VEL
LIN {X 0,Y 256.723,Z 610.961,A -85,B 0,C 180,E1 13244.205,E2 13244.205} C_VEL
LIN {X 0,Y 256.303,Z 616.129,A -85,B 0,C 180,E1 13239.261,E2 13239.261} C_VEL
LIN {X 0,Y 256.41,Z 618.881,A -85,B 0,C 180,E1 13235.147,E2 13235.147} C_VEL
LIN {X 0,Y 256.565,Z 619.998,A -85,B 0,C 180,E1 13231.341,E2 13231.341} C_VEL
LIN {X 0,Y 256.533,Z 619.889,A -85,B 0,C 180,E1 13227.768,E2 13227.768} C_VEL
LIN {X 0,Y 256.366,Z 618.364,A -85,B 0,C 180,E1 13223.957,E2 13223.957} C_VEL
LIN {X 0,Y 256.319,Z 615.357,A -85,B 0,C 180,E1 13219.892,E2 13219.892} C_VEL
LIN {X 0,Y 256.768,Z 610.518,A -85,B 0,C 180,E1 13215.57,E2 13215.57} C_VEL
LIN {X 0,Y 258.051,Z 603.844,A -85,B 0,C 180,E1 13211.242,E2 13211.242} C_VEL
LIN {X 0,Y 260.202,Z 595.782,A -85,B 0,C 180,E1 13207.165,E2 13207.165} C_VEL
LIN {X 0,Y 263.369,Z 585.872,A -85,B 0,C 180,E1 13203.144,E2 13203.144} C_VEL
LIN {X 0,Y 267.627,Z 573.845,A -85,B 0,C 180,E1 13199.216,E2 13199.216} C_VEL
LIN {X 0,Y 272.656,Z 560.199,A -85,B 0,C 180,E1 13195.618,E2 13195.618} C_VEL
LIN {X 0,Y 278.098,Z 545.391,A -85,B 0,C 180,E1 13192.455,E2 13192.455} C_VEL
LIN {X 0,Y 283.488,Z 530.191,A -85,B 0,C 180,E1 13189.803,E2 13189.803} C_VEL
LIN {X 0,Y 288.944,Z 513.87,A -85,B 0,C 180,E1 13187.481,E2 13187.481} C_VEL
LIN {X 0,Y 294.296,Z 496.162,A -85,B 0,C 180,E1 13185.449,E2 13185.449} C_VEL
LIN {X 0,Y 299.398,Z 477.008,A -85,B 0,C 180,E1 13183.712,E2 13183.712} C_VEL
LIN {X 0,Y 303.761,Z 457.692,A -85,B 0,C 180,E1 13182.359,E2 13182.359} C_VEL
LIN {X 0,Y 307.349,Z 438.041,A -85,B 0,C 180,E1 13181.327,E2 13181.327} C_VEL
LIN {X 0,Y 310.084,Z 417.541,A -85,B 0,C 180,E1 13180.555,E2 13180.555} C_VEL
LIN {X 0,Y 312.25,Z 388.031,A -85,B 0,C 180,E1 13179.805,E2 13179.805} C_VEL
LIN {X 0,Y 321.698,Z 235.731,A -85,B 0,C 180,E1 13176.316,E2 13176.316} C_VEL
LIN {X 0,Y 313.353,Z 220.401,A -85,B 0,C 180,E1 13173.807,E2 13173.807} C_VEL
LIN {X 0,Y 305.409,Z 207.37,A -85,B 0,C 180,E1 13171.203,E2 13171.203} C_VEL
LIN {X 0,Y 298.081,Z 196.378,A -85,B 0,C 180,E1 13168.554,E2 13168.554} C_VEL
LIN {X 0,Y 290.945,Z 186.328,A -85,B 0,C 180,E1 13165.658,E2 13165.658} C_VEL
LIN {X 0,Y 285.643,Z 179.404,A -85,B 0,C 180,E1 13163.245,E2 13163.245} C_VEL
LIN {X 0,Y 281.848,Z 174.439,A -85,B 0,C 180,E1 13161.322,E2 13161.322} C_VEL
LIN {X 0,Y 277.061,Z 168.763,A -85,B 0,C 180,E1 13158.625,E2 13158.625} C_VEL
LIN {X 0,Y 275.74,Z 166.891,A -85,B 0,C 180,E1 13157.515,E2 13157.515} C_VEL
LIN {X 0,Y 274.613,Z 164.35,A -85,B 0,C 180,E1 13155.847,E2 13155.847} C_VEL
LIN {X 0,Y 272.332,Z 160.062,A -85,B 0,C 180,E1 13152.295,E2 13152.295} C_VEL
LIN {X 0,Y 269.177,Z 154.333,A -85,B 0,C 180,E1 13144.901,E2 13144.901} C_VEL
LIN {X 0,Y 267.807,Z 153.085,A -85,B 0,C 180,E1 13138.502,E2 13138.502} C_VEL
LIN {X 0,Y 268.343,Z 153.658,A -85,B 0,C 180,E1 13132.721,E2 13132.721} C_VEL
LIN {X 0,Y 269.229,Z 154.7,A -85,B 0,C 180,E1 13129.731,E2 13129.731} C_VEL
LIN {X 0,Y 271.986,Z 159.904,A -85,B 0,C 180,E1 13123.117,E2 13123.117} C_VEL
LIN {X 0,Y 274.55,Z 164.99,A -85,B 0,C 180,E1 13118.866,E2 13118.866} C_VEL
LIN {X 0,Y 276.914,Z 169.746,A -85,B 0,C 180,E1 13115.693,E2 13115.693} C_VEL
LIN {X 0,Y 283.933,Z 178.883,A -85,B 0,C 180,E1 13111.683,E2 13111.683} C_VEL
LIN {X 0,Y 290.914,Z 188.528,A -85,B 0,C 180,E1 13108.447,E2 13108.447} C_VEL
LIN {X 0,Y 298.255,Z 199.235,A -85,B 0,C 180,E1 13105.49,E2 13105.49} C_VEL
LIN {X 0,Y 306.006,Z 211.508,A -85,B 0,C 180,E1 13102.72,E2 13102.72} C_VEL
LIN {X 0,Y 313.808,Z 225.001,A -85,B 0,C 180,E1 13100.205,E2 13100.205} C_VEL
LIN {X 0,Y 320.461,Z 237.88,A -85,B 0,C 180,E1 13098.217,E2 13098.217} C_VEL
LIN {X 0,Y 311.726,Z 397.992,A -85,B 0,C 180,E1 13094.823,E2 13094.823} C_VEL
LIN {X 0,Y 309.58,Z 417.608,A -85,B 0,C 180,E1 13094.113,E2 13094.113} C_VEL
LIN {X 0,Y 306.523,Z 436.654,A -85,B 0,C 180,E1 13093.106,E2 13093.106} C_VEL
LIN {X 0,Y 302.785,Z 454.477,A -85,B 0,C 180,E1 13091.838,E2 13091.838} C_VEL
LIN {X 0,Y 298.187,Z 472.246,A -85,B 0,C 180,E1 13090.2,E2 13090.2} C_VEL
LIN {X 0,Y 293.105,Z 488.869,A -85,B 0,C 180,E1 13088.252,E2 13088.252} C_VEL
LIN {X 0,Y 287.697,Z 504.385,A -85,B 0,C 180,E1 13085.967,E2 13085.967} C_VEL
LIN {X 0,Y 282.113,Z 518.779,A -85,B 0,C 180,E1 13083.32,E2 13083.32} C_VEL
LIN {X 0,Y 276.746,Z 531.593,A -85,B 0,C 180,E1 13080.383,E2 13080.383} C_VEL
LIN {X 0,Y 271.492,Z 543.452,A -85,B 0,C 180,E1 13076.969,E2 13076.969} C_VEL
LIN {X 0,Y 267.02,Z 553.303,A -85,B 0,C 180,E1 13073.384,E2 13073.384} C_VEL
LIN {X 0,Y 263.289,Z 561.591,A -85,B 0,C 180,E1 13069.521,E2 13069.521} C_VEL
LIN {X 0,Y 260.372,Z 568.358,A -85,B 0,C 180,E1 13065.363,E2 13065.363} C_VEL
LIN {X 0,Y 258.365,Z 573.506,A -85,B 0,C 180,E1 13060.93,E2 13060.93} C_VEL
LIN {X 0,Y 257.256,Z 576.818,A -85,B 0,C 180,E1 13056.47,E2 13056.47} C_VEL
LIN {X 0,Y 256.834,Z 578.386,A -85,B 0,C 180,E1 13052.23,E2 13052.23} C_VEL
LIN {X 0,Y 256.819,Z 578.427,A -85,B 0,C 180,E1 13047.991,E2 13047.991} C_VEL
LIN {X 0,Y 257.206,Z 576.98,A -85,B 0,C 180,E1 13043.75,E2 13043.75} C_VEL
LIN {X 0,Y 258.188,Z 573.992,A -85,B 0,C 180,E1 13039.512,E2 13039.512} C_VEL
LIN {X 0,Y 259.959,Z 569.359,A -85,B 0,C 180,E1 13035.293,E2 13035.293} C_VEL
LIN {X 0,Y 262.696,Z 562.943,A -85,B 0,C 180,E1 13031.123,E2 13031.123} C_VEL
LIN {X 0,Y 266.249,Z 555.032,A -85,B 0,C 180,E1 13027.243,E2 13027.243} C_VEL
LIN {X 0,Y 270.508,Z 545.687,A -85,B 0,C 180,E1 13023.668,E2 13023.668} C_VEL
LIN {X 0,Y 275.639,Z 534.209,A -85,B 0,C 180,E1 13020.2,E2 13020.2} C_VEL
LIN {X 0,Y 280.867,Z 521.933,A -85,B 0,C 180,E1 13017.24,E2 13017.24} C_VEL
LIN {X 0,Y 286.526,Z 507.642,A -85,B 0,C 180,E1 13014.477,E2 13014.477} C_VEL
LIN {X 0,Y 292.056,Z 492.21,A -85,B 0,C 180,E1 13012.094,E2 13012.094} C_VEL
LIN {X 0,Y 297.145,Z 476.067,A -85,B 0,C 180,E1 13010.103,E2 13010.103} C_VEL
LIN {X 0,Y 301.899,Z 458.467,A -85,B 0,C 180,E1 13008.39,E2 13008.39} C_VEL
LIN {X 0,Y 305.873,Z 440.482,A -85,B 0,C 180,E1 13007.033,E2 13007.033} C_VEL
LIN {X 0,Y 309.141,Z 421.287,A -85,B 0,C 180,E1 13005.949,E2 13005.949} C_VEL
LIN {X 0,Y 311.474,Z 401.774,A -85,B 0,C 180,E1 13005.185,E2 13005.185} C_VEL
LIN {X 0,Y 313.139,Z 375.952,A -85,B 0,C 180,E1 13004.561,E2 13004.561} C_VEL
LIN {X 0,Y 317.716,Z 289.721,A -85,B 0,C 180,E1 13002.755,E2 13002.755} C_VEL
LIN {X 0,Y 316.791,Z 291.373,A -85,B 0,C 180,E1 13002.61,E2 13002.61} C_VEL
LIN {X 0,Y 314.527,Z 301.164,A -85,B 0,C 180,E1 13002.439,E2 13002.439} C_VEL
LIN {X 0,Y 310.982,Z 324.933,A -85,B 0,C 180,E1 13002.448,E2 13002.448} C_VEL
LIN {X 0,Y 310.034,Z 335.768,A -85,B 0,C 180,E1 13002.6,E2 13002.6} C_VEL
LIN {X 0,Y 306.429,Z 398.583,A -85,B 0,C 180,E1 13003.979,E2 13003.979} C_VEL
LIN {X 0,Y 304.213,Z 418.06,A -85,B 0,C 180,E1 13004.691,E2 13004.691} C_VEL
LIN {X 0,Y 301.171,Z 436.464,A -85,B 0,C 180,E1 13005.665,E2 13005.665} C_VEL
LIN {X 0,Y 297.29,Z 454.4,A -85,B 0,C 180,E1 13006.941,E2 13006.941} C_VEL
LIN {X 0,Y 292.512,Z 472.281,A -85,B 0,C 180,E1 13008.591,E2 13008.591} C_VEL
LIN {X 0,Y 287.225,Z 488.985,A -85,B 0,C 180,E1 13010.556,E2 13010.556} C_VEL
LIN {X 0,Y 281.584,Z 504.575,A -85,B 0,C 180,E1 13012.867,E2 13012.867} C_VEL
LIN {X 0,Y 275.745,Z 519.038,A -85,B 0,C 180,E1 13015.55,E2 13015.55} C_VEL
LIN {X 0,Y 270.113,Z 531.903,A -85,B 0,C 180,E1 13018.537,E2 13018.537} C_VEL
LIN {X 0,Y 264.534,Z 543.919,A -85,B 0,C 180,E1 13022.05,E2 13022.05} C_VEL
LIN {X 0,Y 259.841,Z 553.725,A -85,B 0,C 180,E1 13025.685,E2 13025.685} C_VEL
LIN {X 0,Y 255.776,Z 562.243,A -85,B 0,C 180,E1 13029.751,E2 13029.751} C_VEL
LIN {X 0,Y 252.597,Z 569.156,A -85,B 0,C 180,E1 13034.148,E2 13034.148} C_VEL
LIN {X 0,Y 250.558,Z 574.064,A -85,B 0,C 180,E1 13038.489,E2 13038.489} C_VEL
LIN {X 0,Y 249.344,Z 577.418,A -85,B 0,C 180,E1 13043.089,E2 13043.089} C_VEL
LIN {X 0,Y 248.859,Z 579.052,A -85,B 0,C 180,E1 13047.696,E2 13047.696} C_VEL
LIN {X 0,Y 248.852,Z 579.061,A -85,B 0,C 180,E1 13052.071,E2 13052.071} C_VEL
LIN {X 0,Y 249.277,Z 577.569,A -85,B 0,C 180,E1 13056.447,E2 13056.447} C_VEL
LIN {X 0,Y 250.342,Z 574.538,A -85,B 0,C 180,E1 13060.818,E2 13060.818} C_VEL
LIN {X 0,Y 252.249,Z 569.863,A -85,B 0,C 180,E1 13065.164,E2 13065.164} C_VEL
LIN {X 0,Y 255.171,Z 563.398,A -85,B 0,C 180,E1 13069.453,E2 13069.453} C_VEL
LIN {X 0,Y 258.936,Z 555.437,A -85,B 0,C 180,E1 13073.434,E2 13073.434} C_VEL
LIN {X 0,Y 263.431,Z 546.044,A -85,B 0,C 180,E1 13077.093,E2 13077.093} C_VEL
LIN {X 0,Y 268.476,Z 535.26,A -85,B 0,C 180,E1 13080.429,E2 13080.429} C_VEL
LIN {X 0,Y 274.287,Z 522.184,A -85,B 0,C 180,E1 13083.646,E2 13083.646} C_VEL
LIN {X 0,Y 280.128,Z 507.991,A -85,B 0,C 180,E1 13086.423,E2 13086.423} C_VEL
LIN {X 0,Y 285.73,Z 492.924,A -85,B 0,C 180,E1 13088.781,E2 13088.781} C_VEL
LIN {X 0,Y 291.165,Z 476.297,A -85,B 0,C 180,E1 13090.855,E2 13090.855} C_VEL
LIN {X 0,Y 295.891,Z 459.416,A -85,B 0,C 180,E1 13092.517,E2 13092.517} C_VEL
LIN {X 0,Y 300,Z 441.601,A -85,B 0,C 180,E1 13093.885,E2 13093.885} C_VEL
LIN {X 0,Y 303.401,Z 422.538,A -85,B 0,C 180,E1 13094.985,E2 13094.985} C_VEL
LIN {X 0,Y 305.904,Z 402.619,A -85,B 0,C 180,E1 13095.783,E2 13095.783} C_VEL
LIN {X 0,Y 307.668,Z 376.716,A -85,B 0,C 180,E1 13096.421,E2 13096.421} C_VEL
LIN {X 0,Y 315.211,Z 240.935,A -85,B 0,C 180,E1 13099.306,E2 13099.306} C_VEL
LIN {X 0,Y 307.251,Z 225.691,A -85,B 0,C 180,E1 13101.837,E2 13101.837} C_VEL
LIN {X 0,Y 299.361,Z 212.414,A -85,B 0,C 180,E1 13104.585,E2 13104.585} C_VEL
LIN {X 0,Y 292.476,Z 201.64,A -85,B 0,C 180,E1 13107.265,E2 13107.265} C_VEL
LIN {X 0,Y 286.871,Z 193.49,A -85,B 0,C 180,E1 13109.701,E2 13109.701} C_VEL
LIN {X 0,Y 283.828,Z 189.267,A -85,B 0,C 180,E1 13111.143,E2 13111.143} C_VEL
LIN {X 0,Y 279.964,Z 183.951,A -85,B 0,C 180,E1 13113.142,E2 13113.142} C_VEL
LIN {X 0,Y 273.703,Z 175.795,A -85,B 0,C 180,E1 13116.877,E2 13116.877} C_VEL
LIN {X 0,Y 269.36,Z 170.328,A -85,B 0,C 180,E1 13120.031,E2 13120.031} C_VEL
LIN {X 0,Y 267.13,Z 165.81,A -85,B 0,C 180,E1 13123.92,E2 13123.92} C_VEL
LIN {X 0,Y 264.653,Z 160.925,A -85,B 0,C 180,E1 13130.65,E2 13130.65} C_VEL
LIN {X 0,Y 263.521,Z 159.847,A -85,B 0,C 180,E1 13136.737,E2 13136.737} C_VEL
LIN {X 0,Y 264.069,Z 160.402,A -85,B 0,C 180,E1 13142.387,E2 13142.387} C_VEL
LIN {X 0,Y 265.081,Z 161.51,A -85,B 0,C 180,E1 13145.628,E2 13145.628} C_VEL
LIN {X 0,Y 267.825,Z 166.604,A -85,B 0,C 180,E1 13152.067,E2 13152.067} C_VEL
LIN {X 0,Y 268.745,Z 168.712,A -85,B 0,C 180,E1 13153.555,E2 13153.555} C_VEL
LIN {X 0,Y 272.396,Z 172.81,A -85,B 0,C 180,E1 13156.308,E2 13156.308} C_VEL
LIN {X 0,Y 276.946,Z 178.393,A -85,B 0,C 180,E1 13159.234,E2 13159.234} C_VEL
LIN {X 0,Y 280.915,Z 183.327,A -85,B 0,C 180,E1 13161.451,E2 13161.451} C_VEL
LIN {X 0,Y 285.778,Z 189.855,A -85,B 0,C 180,E1 13163.889,E2 13163.889} C_VEL
LIN {X 0,Y 292.108,Z 198.663,A -85,B 0,C 180,E1 13166.696,E2 13166.696} C_VEL
LIN {X 0,Y 299.759,Z 209.978,A -85,B 0,C 180,E1 13169.691,E2 13169.691} C_VEL
LIN {X 0,Y 307.758,Z 223.194,A -85,B 0,C 180,E1 13172.498,E2 13172.498} C_VEL
LIN {X 0,Y 315.572,Z 237.417,A -85,B 0,C 180,E1 13174.993,E2 13174.993} C_VEL
LIN {X 0,Y 316.538,Z 239.517,A -85,B 0,C 180,E1 13175.297,E2 13175.297} C_VEL
LIN {X 0,Y 305.095,Z 413.574,A -85,B 0,C 180,E1 13179.331,E2 13179.331} C_VEL
LIN {X 0,Y 302.31,Z 435.117,A -85,B 0,C 180,E1 13180.101,E2 13180.101} C_VEL
LIN {X 0,Y 298.493,Z 455.892,A -85,B 0,C 180,E1 13181.165,E2 13181.165} C_VEL
LIN {X 0,Y 293.854,Z 475.898,A -85,B 0,C 180,E1 13182.555,E2 13182.555} C_VEL
LIN {X 0,Y 288.525,Z 495.25,A -85,B 0,C 180,E1 13184.309,E2 13184.309} C_VEL
LIN {X 0,Y 282.796,Z 513.483,A -85,B 0,C 180,E1 13186.416,E2 13186.416} C_VEL
LIN {X 0,Y 276.814,Z 530.645,A -85,B 0,C 180,E1 13188.901,E2 13188.901} C_VEL
LIN {X 0,Y 271.011,Z 546.208,A -85,B 0,C 180,E1 13191.699,E2 13191.699} C_VEL
LIN {X 0,Y 265.53,Z 560.347,A -85,B 0,C 180,E1 13194.824,E2 13194.824} C_VEL
LIN {X 0,Y 260.542,Z 573.13,A -85,B 0,C 180,E1 13198.283,E2 13198.283} C_VEL
LIN {X 0,Y 256.007,Z 585.173,A -85,B 0,C 180,E1 13202.307,E2 13202.307} C_VEL
LIN {X 0,Y 252.448,Z 595.586,A -85,B 0,C 180,E1 13206.669,E2 13206.669} C_VEL
LIN {X 0,Y 250.073,Z 603.932,A -85,B 0,C 180,E1 13211.105,E2 13211.105} C_VEL
LIN {X 0,Y 248.753,Z 610.473,A -85,B 0,C 180,E1 13215.624,E2 13215.624} C_VEL
LIN {X 0,Y 248.322,Z 615.14,A -85,B 0,C 180,E1 13220.031,E2 13220.031} C_VEL
LIN {X 0,Y 248.395,Z 617.966,A -85,B 0,C 180,E1 13224.226,E2 13224.226} C_VEL
LIN {X 0,Y 248.573,Z 619.297,A -85,B 0,C 180,E1 13228.157,E2 13228.157} C_VEL
LIN {X 0,Y 248.581,Z 619.326,A -85,B 0,C 180,E1 13231.615,E2 13231.615} C_VEL
LIN {X 0,Y 248.408,Z 618.105,A -85,B 0,C 180,E1 13235.545,E2 13235.545} C_VEL
LIN {X 0,Y 248.316,Z 615.339,A -85,B 0,C 180,E1 13239.738,E2 13239.738} C_VEL
LIN {X 0,Y 248.909,Z 610.165,A -85,B 0,C 180,E1 13245.137,E2 13245.137} C_VEL
LIN {X 0,Y 250.434,Z 604.152,A -85,B 0,C 180,E1 13249.597,E2 13249.597} C_VEL
LIN {X 0,Y 253.295,Z 595.945,A -85,B 0,C 180,E1 13254.24,E2 13254.24} C_VEL
LIN {X 0,Y 257.841,Z 585.31,A -85,B 0,C 180,E1 13258.996,E2 13258.996} C_VEL
LIN {X 0,Y 264.12,Z 572.545,A -85,B 0,C 180,E1 13263.554,E2 13263.554} C_VEL
LIN {X 0,Y 272.704,Z 557.041,A -85,B 0,C 180,E1 13268.024,E2 13268.024} C_VEL
LIN {X 0,Y 282.388,Z 541.123,A -85,B 0,C 180,E1 13271.734,E2 13271.734} C_VEL
LIN {X 0,Y 293.929,Z 523.511,A -85,B 0,C 180,E1 13275.038,E2 13275.038} C_VEL
LIN {X 0,Y 307.79,Z 503.202,A -85,B 0,C 180,E1 13277.928,E2 13277.928} C_VEL
LIN {X 0,Y 308.787,Z 501.73,A -85,B 0,C 180,E1 13278.131,E2 13278.131} C_VEL
LIN {X 0,Y 298.828,Z 517.354,A -85,B 0,C 180,E1 13280.527,E2 13280.527} C_VEL
LIN {X 0,Y 288.871,Z 532.258,A -85,B 0,C 180,E1 13283.464,E2 13283.464} C_VEL
LIN {X 0,Y 280.134,Z 544.99,A -85,B 0,C 180,E1 13286.657,E2 13286.657} C_VEL
LIN {X 0,Y 272.542,Z 555.625,A -85,B 0,C 180,E1 13290.071,E2 13290.071} C_VEL
LIN {X 0,Y 265.753,Z 564.76,A -85,B 0,C 180,E1 13293.884,E2 13293.884} C_VEL
LIN {X 0,Y 260.214,Z 571.895,A -85,B 0,C 180,E1 13297.88,E2 13297.88} C_VEL
LIN {X 0,Y 255.898,Z 577.126,A -85,B 0,C 180,E1 13302.021,E2 13302.021} C_VEL
LIN {X 0,Y 252.731,Z 580.458,A -85,B 0,C 180,E1 13306.269,E2 13306.269} C_VEL
LIN {X 0,Y 250.624,Z 581.941,A -85,B 0,C 180,E1 13310.586,E2 13310.586} C_VEL
LIN {X 0,Y 249.445,Z 581.663,A -85,B 0,C 180,E1 13314.711,E2 13314.711} C_VEL
LIN {X 0,Y 248.891,Z 579.862,A -85,B 0,C 180,E1 13318.619,E2 13318.619} C_VEL
LIN {X 0,Y 248.699,Z 576.493,A -85,B 0,C 180,E1 13322.535,E2 13322.535} C_VEL
LIN {X 0,Y 248.816,Z 571.459,A -85,B 0,C 180,E1 13326.461,E2 13326.461} C_VEL
LIN {X 0,Y 249.281,Z 565.095,A -85,B 0,C 180,E1 13330.165,E2 13330.165} C_VEL
LIN {X 0,Y 250.186,Z 556.903,A -85,B 0,C 180,E1 13333.874,E2 13333.874} C_VEL
LIN {X 0,Y 251.644,Z 546.678,A -85,B 0,C 180,E1 13337.577,E2 13337.577} C_VEL
LIN {X 0,Y 253.568,Z 534.971,A -85,B 0,C 180,E1 13341.029,E2 13341.029} C_VEL
LIN {X 0,Y 255.905,Z 521.808,A -85,B 0,C 180,E1 13344.221,E2 13344.221} C_VEL
LIN {X 0,Y 258.639,Z 506.719,A -85,B 0,C 180,E1 13347.232,E2 13347.232} C_VEL
LIN {X 0,Y 261.553,Z 490.11,A -85,B 0,C 180,E1 13349.926,E2 13349.926} C_VEL
LIN {X 0,Y 264.544,Z 471.788,A -85,B 0,C 180,E1 13352.331,E2 13352.331} C_VEL
LIN {X 0,Y 267.256,Z 453.384,A -85,B 0,C 180,E1 13354.267,E2 13354.267} C_VEL
LIN {X 0,Y 269.672,Z 434.041,A -85,B 0,C 180,E1 13355.861,E2 13355.861} C_VEL
LIN {X 0,Y 270.855,Z 422.936,A -85,B 0,C 180,E1 13356.597,E2 13356.597} C_VEL
LIN {X 0,Y 271.591,Z 423.385,A -85,B 0,C 180,E1 13356.876,E2 13356.876} C_VEL
LIN {X 0,Y 273.362,Z 422.414,A -85,B 0,C 180,E1 13357.32,E2 13357.32} C_VEL
LIN {X 0,Y 276.438,Z 418.48,A -85,B 0,C 180,E1 13357.845,E2 13357.845} C_VEL
LIN {X 0,Y 280.752,Z 409.49,A -85,B 0,C 180,E1 13358.342,E2 13358.342} C_VEL
LIN {X 0,Y 283.669,Z 400.971,A -85,B 0,C 180,E1 13358.6,E2 13358.6} C_VEL
LIN {X 0,Y 286.446,Z 397.274,A -85,B 0,C 180,E1 13359.151,E2 13359.151} C_VEL
LIN {X 0,Y 289.538,Z 390.375,A -85,B 0,C 180,E1 13359.65,E2 13359.65} C_VEL
LIN {X 0,Y 294.23,Z 374.759,A -85,B 0,C 180,E1 13360.256,E2 13360.256} C_VEL
LIN {X 0,Y 298.61,Z 357.239,A -85,B 0,C 180,E1 13360.7,E2 13360.7} C_VEL
LIN {X 0,Y 301.961,Z 351.159,A -85,B 0,C 180,E1 13361.288,E2 13361.288} C_VEL
LIN {X 0,Y 305.971,Z 340.385,A -85,B 0,C 180,E1 13361.845,E2 13361.845} C_VEL
LIN {X 0,Y 310.687,Z 324.049,A -85,B 0,C 180,E1 13362.354,E2 13362.354} C_VEL
LIN {X 0,Y 310.034,Z 335.768,A -85,B 0,C 180,E1 13362.6,E2 13362.6} C_VEL
LIN {X 0,Y 309.114,Z 342.591,A -85,B 0,C 180,E1 13362.625,E2 13362.625} C_VEL
LIN {X 0,Y 306.373,Z 352.513,A -85,B 0,C 180,E1 13362.349,E2 13362.349} C_VEL
LIN {X 0,Y 300.9,Z 368.892,A -85,B 0,C 180,E1 13361.661,E2 13361.661} C_VEL
LIN {X 0,Y 300.303,Z 371.146,A -85,B 0,C 180,E1 13361.6,E2 13361.6} C_VEL
LIN {X 0,Y 295.203,Z 389.251,A -85,B 0,C 180,E1 13361.03,E2 13361.03} C_VEL
LIN {X 0,Y 291.421,Z 398.857,A -85,B 0,C 180,E1 13360.523,E2 13360.523} C_VEL
LIN {X 0,Y 287.742,Z 404.824,A -85,B 0,C 180,E1 13359.94,E2 13359.94} C_VEL
LIN {X 0,Y 286.745,Z 406.485,A -85,B 0,C 180,E1 13359.781,E2 13359.781} C_VEL
LIN {X 0,Y 282.933,Z 416.142,A -85,B 0,C 180,E1 13359.486,E2 13359.486} C_VEL
LIN {X 0,Y 278.498,Z 424.056,A -85,B 0,C 180,E1 13358.99,E2 13358.99} C_VEL
LIN {X 0,Y 274.713,Z 428.545,A -85,B 0,C 180,E1 13358.358,E2 13358.358} C_VEL
LIN {X 0,Y 272.206,Z 430.447,A -85,B 0,C 180,E1 13357.838,E2 13357.838} C_VEL
LIN {X 0,Y 267.787,Z 437.538,A -85,B 0,C 180,E1 13357.368,E2 13357.368} C_VEL
LIN {X 0,Y 264.841,Z 440.803,A -85,B 0,C 180,E1 13356.89,E2 13356.89} C_VEL
LIN {X 0,Y 262.747,Z 442.191,A -85,B 0,C 180,E1 13356.416,E2 13356.416} C_VEL
LIN {X 0,Y 261.266,Z 442.173,A -85,B 0,C 180,E1 13355.875,E2 13355.875} C_VEL
LIN {X 0,Y 258.539,Z 461.784,A -85,B 0,C 180,E1 13354.038,E2 13354.038} C_VEL
LIN {X 0,Y 255.636,Z 479.949,A -85,B 0,C 180,E1 13351.872,E2 13351.872} C_VEL
LIN {X 0,Y 252.564,Z 497.58,A -85,B 0,C 180,E1 13349.27,E2 13349.27} C_VEL
LIN {X 0,Y 249.653,Z 513.477,A -85,B 0,C 180,E1 13346.395,E2 13346.395} C_VEL
LIN {X 0,Y 247.013,Z 527.786,A -85,B 0,C 180,E1 13343.239,E2 13343.239} C_VEL
LIN {X 0,Y 244.76,Z 540.472,A -85,B 0,C 180,E1 13339.82,E2 13339.82} C_VEL
LIN {X 0,Y 243.017,Z 551.359,A -85,B 0,C 180,E1 13336.247,E2 13336.247} C_VEL
LIN {X 0,Y 241.759,Z 560.774,A -85,B 0,C 180,E1 13332.42,E2 13332.42} C_VEL
LIN {X 0,Y 241.008,Z 568.701,A -85,B 0,C 180,E1 13328.35,E2 13328.35} C_VEL
LIN {X 0,Y 240.714,Z 574.732,A -85,B 0,C 180,E1 13324.288,E2 13324.288} C_VEL
LIN {X 0,Y 240.786,Z 578.995,A -85,B 0,C 180,E1 13320.238,E2 13320.238} C_VEL
LIN {X 0,Y 241.193,Z 581.676,A -85,B 0,C 180,E1 13316.197,E2 13316.197} C_VEL
LIN {X 0,Y 242.18,Z 582.869,A -85,B 0,C 180,E1 13311.931,E2 13311.931} C_VEL
LIN {X 0,Y 243.947,Z 582.407,A -85,B 0,C 180,E1 13307.695,E2 13307.695} C_VEL
LIN {X 0,Y 246.853,Z 580.181,A -85,B 0,C 180,E1 13303.287,E2 13303.287} C_VEL
LIN {X 0,Y 250.957,Z 576.159,A -85,B 0,C 180,E1 13298.988,E2 13298.988} C_VEL
LIN {X 0,Y 256.316,Z 570.236,A -85,B 0,C 180,E1 13294.826,E2 13294.826} C_VEL
LIN {X 0,Y 262.936,Z 562.472,A -85,B 0,C 180,E1 13290.874,E2 13290.874} C_VEL
LIN {X 0,Y 271.332,Z 552.193,A -85,B 0,C 180,E1 13286.95,E2 13286.95} C_VEL
LIN {X 0,Y 280.128,Z 540.972,A -85,B 0,C 180,E1 13283.666,E2 13283.666} C_VEL
LIN {X 0,Y 290.701,Z 526.969,A -85,B 0,C 180,E1 13280.484,E2 13280.484} C_VEL
LIN {X 0,Y 300.036,Z 514.245,A -85,B 0,C 180,E1 13278.204,E2 13278.204} C_VEL
LIN {X 0,Y 289.144,Z 528.517,A -85,B 0,C 180,E1 13275.995,E2 13275.995} C_VEL
LIN {X 0,Y 275.924,Z 546.438,A -85,B 0,C 180,E1 13272.378,E2 13272.378} C_VEL
LIN {X 0,Y 265.329,Z 561.943,A -85,B 0,C 180,E1 13268.389,E2 13268.389} C_VEL
LIN {X 0,Y 256.18,Z 576.722,A -85,B 0,C 180,E1 13263.658,E2 13263.658} C_VEL
LIN {X 0,Y 249.501,Z 588.946,A -85,B 0,C 180,E1 13258.745,E2 13258.745} C_VEL
LIN {X 0,Y 244.964,Z 598.59,A -85,B 0,C 180,E1 13253.835,E2 13253.835} C_VEL
LIN {X 0,Y 242.155,Z 605.985,A -85,B 0,C 180,E1 13248.997,E2 13248.997} C_VEL
LIN {X 0,Y 240.755,Z 611.204,A -85,B 0,C 180,E1 13244.431,E2 13244.431} C_VEL
LIN {X 0,Y 240.323,Z 615.75,A -85,B 0,C 180,E1 13238.616,E2 13238.616} C_VEL
LIN {X 0,Y 240.49,Z 618.033,A -85,B 0,C 180,E1 13234.293,E2 13234.293} C_VEL
LIN {X 0,Y 240.63,Z 618.808,A -85,B 0,C 180,E1 13230.478,E2 13230.478} C_VEL
LIN {X 0,Y 240.527,Z 618.256,A -85,B 0,C 180,E1 13226.427,E2 13226.427} C_VEL
LIN {X 0,Y 240.343,Z 616.42,A -85,B 0,C 180,E1 13222.351,E2 13222.351} C_VEL
LIN {X 0,Y 240.44,Z 612.898,A -85,B 0,C 180,E1 13218.001,E2 13218.001} C_VEL
LIN {X 0,Y 241.269,Z 607.55,A -85,B 0,C 180,E1 13213.386,E2 13213.386} C_VEL
LIN {X 0,Y 243.106,Z 600.411,A -85,B 0,C 180,E1 13208.783,E2 13208.783} C_VEL
LIN {X 0,Y 245.946,Z 591.88,A -85,B 0,C 180,E1 13204.475,E2 13204.475} C_VEL
LIN {X 0,Y 249.982,Z 581.29,A -85,B 0,C 180,E1 13200.219,E2 13200.219} C_VEL
LIN {X 0,Y 255.087,Z 568.706,A -85,B 0,C 180,E1 13196.181,E2 13196.181} C_VEL
LIN {X 0,Y 260.651,Z 555.205,A -85,B 0,C 180,E1 13192.695,E2 13192.695} C_VEL
LIN {X 0,Y 266.874,Z 539.718,A -85,B 0,C 180,E1 13189.473,E2 13189.473} C_VEL
LIN {X 0,Y 273.242,Z 522.95,A -85,B 0,C 180,E1 13186.679,E2 13186.679} C_VEL
LIN {X 0,Y 279.183,Z 505.877,A -85,B 0,C 180,E1 13184.407,E2 13184.407} C_VEL
LIN {X 0,Y 284.772,Z 487.896,A -85,B 0,C 180,E1 13182.498,E2 13182.498} C_VEL
LIN {X 0,Y 289.825,Z 469.137,A -85,B 0,C 180,E1 13180.931,E2 13180.931} C_VEL
LIN {X 0,Y 294.201,Z 449.631,A -85,B 0,C 180,E1 13179.684,E2 13179.684} C_VEL
LIN {X 0,Y 297.862,Z 428.81,A -85,B 0,C 180,E1 13178.719,E2 13178.719} C_VEL
LIN {X 0,Y 300.33,Z 407.261,A -85,B 0,C 180,E1 13178.024,E2 13178.024} C_VEL
LIN {X 0,Y 311.367,Z 242.66,A -85,B 0,C 180,E1 13174.191,E2 13174.191} C_VEL
LIN {X 0,Y 303.105,Z 227.255,A -85,B 0,C 180,E1 13171.412,E2 13171.412} C_VEL
LIN {X 0,Y 295.4,Z 214.632,A -85,B 0,C 180,E1 13168.561,E2 13168.561} C_VEL
LIN {X 0,Y 287.646,Z 202.823,A -85,B 0,C 180,E1 13165.312,E2 13165.312} C_VEL
LIN {X 0,Y 281.063,Z 193.757,A -85,B 0,C 180,E1 13162.153,E2 13162.153} C_VEL
LIN {X 0,Y 277.187,Z 188.572,A -85,B 0,C 180,E1 13160.04,E2 13160.04} C_VEL
LIN {X 0,Y 273.012,Z 183.279,A -85,B 0,C 180,E1 13157.476,E2 13157.476} C_VEL
LIN {X 0,Y 269.436,Z 178.896,A -85,B 0,C 180,E1 13154.946,E2 13154.946} C_VEL
LIN {X 0,Y 265.227,Z 173.675,A -85,B 0,C 180,E1 13151.305,E2 13151.305} C_VEL
LIN {X 0,Y 260.901,Z 168.756,A -85,B 0,C 180,E1 13146.049,E2 13146.049} C_VEL
LIN {X 0,Y 260.399,Z 167.696,A -85,B 0,C 180,E1 13144.404,E2 13144.404} C_VEL
LIN {X 0,Y 259.228,Z 166.596,A -85,B 0,C 180,E1 13138.231,E2 13138.231} C_VEL
LIN {X 0,Y 259.778,Z 167.196,A -85,B 0,C 180,E1 13132.48,E2 13132.48} C_VEL
LIN {X 0,Y 260.448,Z 168.001,A -85,B 0,C 180,E1 13130.051,E2 13130.051} C_VEL
LIN {X 0,Y 261.262,Z 170.227,A -85,B 0,C 180,E1 13127.386,E2 13127.386} C_VEL
LIN {X 0,Y 264.459,Z 173.862,A -85,B 0,C 180,E1 13123.527,E2 13123.527} C_VEL
LIN {X 0,Y 268.786,Z 179.241,A -85,B 0,C 180,E1 13119.646,E2 13119.646} C_VEL
LIN {X 0,Y 273.434,Z 185.298,A -85,B 0,C 180,E1 13116.339,E2 13116.339} C_VEL
LIN {X 0,Y 279.553,Z 193.475,A -85,B 0,C 180,E1 13112.754,E2 13112.754} C_VEL
LIN {X 0,Y 284.647,Z 200.85,A -85,B 0,C 180,E1 13110.18,E2 13110.18} C_VEL
LIN {X 0,Y 291.02,Z 210.286,A -85,B 0,C 180,E1 13107.356,E2 13107.356} C_VEL
LIN {X 0,Y 298.972,Z 223.444,A -85,B 0,C 180,E1 13104.237,E2 13104.237} C_VEL
LIN {X 0,Y 306.295,Z 236.714,A -85,B 0,C 180,E1 13101.667,E2 13101.667} C_VEL
LIN {X 0,Y 310.221,Z 244.789,A -85,B 0,C 180,E1 13100.369,E2 13100.369} C_VEL
LIN {X 0,Y 301.079,Z 398.476,A -85,B 0,C 180,E1 13097.057,E2 13097.057} C_VEL
LIN {X 0,Y 298.762,Z 418.237,A -85,B 0,C 180,E1 13096.334,E2 13096.334} C_VEL
LIN {X 0,Y 295.555,Z 436.973,A -85,B 0,C 180,E1 13095.336,E2 13095.336} C_VEL
LIN {X 0,Y 291.412,Z 455.404,A -85,B 0,C 180,E1 13094.009,E2 13094.009} C_VEL
LIN {X 0,Y 286.476,Z 473.16,A -85,B 0,C 180,E1 13092.344,E2 13092.344} C_VEL
LIN {X 0,Y 281.006,Z 489.79,A -85,B 0,C 180,E1 13090.357,E2 13090.357} C_VEL
LIN {X 0,Y 275.16,Z 505.326,A -85,B 0,C 180,E1 13088.017,E2 13088.017} C_VEL
LIN {X 0,Y 269.304,Z 519.274,A -85,B 0,C 180,E1 13085.392,E2 13085.392} C_VEL
LIN {X 0,Y 263.418,Z 532.192,A -85,B 0,C 180,E1 13082.355,E2 13082.355} C_VEL
LIN {X 0,Y 257.57,Z 544.275,A -85,B 0,C 180,E1 13078.772,E2 13078.772} C_VEL
LIN {X 0,Y 252.363,Z 554.631,A -85,B 0,C 180,E1 13074.831,E2 13074.831} C_VEL
LIN {X 0,Y 248.21,Z 562.907,A -85,B 0,C 180,E1 13070.76,E2 13070.76} C_VEL
LIN {X 0,Y 244.932,Z 569.663,A -85,B 0,C 180,E1 13066.358,E2 13066.358} C_VEL
LIN {X 0,Y 242.651,Z 574.804,A -85,B 0,C 180,E1 13061.647,E2 13061.647} C_VEL
LIN {X 0,Y 241.38,Z 578.111,A -85,B 0,C 180,E1 13056.898,E2 13056.898} C_VEL
LIN {X 0,Y 240.893,Z 579.677,A -85,B 0,C 180,E1 13052.377,E2 13052.377} C_VEL
LIN {X 0,Y 240.877,Z 579.717,A -85,B 0,C 180,E1 13047.858,E2 13047.858} C_VEL
LIN {X 0,Y 241.324,Z 578.273,A -85,B 0,C 180,E1 13043.337,E2 13043.337} C_VEL
LIN {X 0,Y 242.453,Z 575.289,A -85,B 0,C 180,E1 13038.822,E2 13038.822} C_VEL
LIN {X 0,Y 244.471,Z 570.661,A -85,B 0,C 180,E1 13034.338,E2 13034.338} C_VEL
LIN {X 0,Y 247.554,Z 564.252,A -85,B 0,C 180,E1 13029.92,E2 13029.92} C_VEL
LIN {X 0,Y 251.516,Z 556.354,A -85,B 0,C 180,E1 13025.828,E2 13025.828} C_VEL
LIN {X 0,Y 256.53,Z 546.419,A -85,B 0,C 180,E1 13021.86,E2 13021.86} C_VEL
LIN {X 0,Y 261.852,Z 535.579,A -85,B 0,C 180,E1 13018.457,E2 13018.457} C_VEL
LIN {X 0,Y 267.548,Z 523.346,A -85,B 0,C 180,E1 13015.385,E2 13015.385} C_VEL
LIN {X 0,Y 273.684,Z 509.114,A -85,B 0,C 180,E1 13012.533,E2 13012.533} C_VEL
LIN {X 0,Y 279.763,Z 493.446,A -85,B 0,C 180,E1 13010.04,E2 13010.04} C_VEL
LIN {X 0,Y 285.313,Z 477.139,A -85,B 0,C 180,E1 13007.982,E2 13007.982} C_VEL
LIN {X 0,Y 290.475,Z 459.362,A -85,B 0,C 180,E1 13006.22,E2 13006.22} C_VEL
LIN {X 0,Y 294.735,Z 441.409,A -85,B 0,C 180,E1 13004.844,E2 13004.844} C_VEL
LIN {X 0,Y 298.288,Z 421.975,A -85,B 0,C 180,E1 13003.732,E2 13003.732} C_VEL
LIN {X 0,Y 300.806,Z 402.344,A -85,B 0,C 180,E1 13002.954,E2 13002.954} C_VEL
LIN {X 0,Y 302.636,Z 376.109,A -85,B 0,C 180,E1 13002.31,E2 13002.31} C_VEL
LIN {X 0,Y 303.464,Z 360.04,A -85,B 0,C 180,E1 13001.947,E2 13001.947} C_VEL
LIN {X 0,Y 302.475,Z 362.063,A -85,B 0,C 180,E1 13001.789,E2 13001.789} C_VEL
LIN {X 0,Y 300.303,Z 371.146,A -85,B 0,C 180,E1 13001.6,E2 13001.6} C_VEL
LIN {X 0,Y 293.618,Z 400.26,A -85,B 0,C 180,E1 13001.149,E2 13001.149} C_VEL
LIN {X 0,Y 290.117,Z 411.398,A -85,B 0,C 180,E1 13000.99,E2 13000.99} C_VEL
LIN {X 0,Y 285.817,Z 421.089,A -85,B 0,C 180,E1 13000.676,E2 13000.676} C_VEL
LIN {X 0,Y 281.198,Z 428.764,A -85,B 0,C 180,E1 13000.193,E2 13000.193} C_VEL
LIN {X 0,Y 276.531,Z 434.042,A -85,B 0,C 180,E1 12999.522,E2 12999.522} C_VEL
LIN {X 0,Y 274.251,Z 435.964,A -85,B 0,C 180,E1 12999.104,E2 12999.104} C_VEL
LIN {X 0,Y 269.293,Z 443.017,A -85,B 0,C 180,E1 12998.592,E2 12998.592} C_VEL
LIN {X 0,Y 265.135,Z 447.196,A -85,B 0,C 180,E1 12997.93,E2 12997.93} C_VEL
LIN {X 0,Y 261.371,Z 449.616,A -85,B 0,C 180,E1 12997.119,E2 12997.119} C_VEL
LIN {X 0,Y 256.937,Z 454.705,A -85,B 0,C 180,E1 12996.541,E2 12996.541} C_VEL
LIN {X 0,Y 253.939,Z 456.992,A -85,B 0,C 180,E1 12995.922,E2 12995.922} C_VEL
LIN {X 0,Y 252.193,Z 457.362,A -85,B 0,C 180,E1 12995.37,E2 12995.37} C_VEL
LIN {X 0,Y 251.716,Z 457.168,A -85,B 0,C 180,E1 12995.132,E2 12995.132} C_VEL
LIN {X 0,Y 248.612,Z 476.661,A -85,B 0,C 180,E1 12992.884,E2 12992.884} C_VEL
LIN {X 0,Y 245.497,Z 494.338,A -85,B 0,C 180,E1 12990.334,E2 12990.334} C_VEL
LIN {X 0,Y 242.399,Z 510.848,A -85,B 0,C 180,E1 12987.384,E2 12987.384} C_VEL
LIN {X 0,Y 239.579,Z 525.651,A -85,B 0,C 180,E1 12984.142,E2 12984.142} C_VEL
LIN {X 0,Y 237.145,Z 538.896,A -85,B 0,C 180,E1 12980.606,E2 12980.606} C_VEL
LIN {X 0,Y 235.21,Z 550.528,A -85,B 0,C 180,E1 12976.802,E2 12976.802} C_VEL
LIN {X 0,Y 233.855,Z 560.269,A -85,B 0,C 180,E1 12972.846,E2 12972.846} C_VEL
LIN {X 0,Y 233.071,Z 568.078,A -85,B 0,C 180,E1 12968.885,E2 12968.885} C_VEL
LIN {X 0,Y 232.725,Z 574.434,A -85,B 0,C 180,E1 12964.683,E2 12964.683} C_VEL
LIN {X 0,Y 232.778,Z 579.058,A -85,B 0,C 180,E1 12960.493,E2 12960.493} C_VEL
LIN {X 0,Y 233.184,Z 582.085,A -85,B 0,C 180,E1 12956.313,E2 12956.313} C_VEL
LIN {X 0,Y 234.204,Z 583.634,A -85,B 0,C 180,E1 12951.902,E2 12951.902} C_VEL
LIN {X 0,Y 236.184,Z 583.494,A -85,B 0,C 180,E1 12947.283,E2 12947.283} C_VEL
LIN {X 0,Y 239.299,Z 581.589,A -85,B 0,C 180,E1 12942.744,E2 12942.744} C_VEL
LIN {X 0,Y 243.679,Z 577.927,A -85,B 0,C 180,E1 12938.329,E2 12938.329} C_VEL
LIN {X 0,Y 249.717,Z 572.185,A -85,B 0,C 180,E1 12933.869,E2 12933.869} C_VEL
LIN {X 0,Y 256.819,Z 564.851,A -85,B 0,C 180,E1 12929.853,E2 12929.853} C_VEL
LIN {X 0,Y 265.731,Z 555.1,A -85,B 0,C 180,E1 12925.901,E2 12925.901} C_VEL
LIN {X 0,Y 276.151,Z 543.291,A -85,B 0,C 180,E1 12922.274,E2 12922.274} C_VEL
LIN {X 0,Y 287.423,Z 529.971,A -85,B 0,C 180,E1 12919.157,E2 12919.157} C_VEL
LIN {X 0,Y 290.874,Z 525.828,A -85,B 0,C 180,E1 12918.314,E2 12918.314} C_VEL
LIN {X 0,Y 278.534,Z 540.359,A -85,B 0,C 180,E1 12915.592,E2 12915.592} C_VEL
LIN {X 0,Y 266.144,Z 555.686,A -85,B 0,C 180,E1 12911.97,E2 12911.97} C_VEL
LIN {X 0,Y 254.978,Z 570.715,A -85,B 0,C 180,E1 12907.433,E2 12907.433} C_VEL
LIN {X 0,Y 246.468,Z 583.296,A -85,B 0,C 180,E1 12902.654,E2 12902.654} C_VEL
LIN {X 0,Y 240.069,Z 594.061,A -85,B 0,C 180,E1 12897.487,E2 12897.487} C_VEL
LIN {X 0,Y 235.781,Z 602.676,A -85,B 0,C 180,E1 12892.175,E2 12892.175} C_VEL
LIN {X 0,Y 233.451,Z 608.753,A -85,B 0,C 180,E1 12887.19,E2 12887.19} C_VEL
LIN {X 0,Y 232.443,Z 613.009,A -85,B 0,C 180,E1 12882.169,E2 12882.169} C_VEL
LIN {X 0,Y 232.412,Z 616.565,A -85,B 0,C 180,E1 12876.396,E2 12876.396} C_VEL
LIN {X 0,Y 232.607,Z 617.981,A -85,B 0,C 180,E1 12872.219,E2 12872.219} C_VEL
LIN {X 0,Y 232.636,Z 618.059,A -85,B 0,C 180,E1 12868.524,E2 12868.524} C_VEL
LIN {X 0,Y 232.435,Z 616.917,A -85,B 0,C 180,E1 12864.324,E2 12864.324} C_VEL
LIN {X 0,Y 232.345,Z 614.186,A -85,B 0,C 180,E1 12859.839,E2 12859.839} C_VEL
LIN {X 0,Y 232.852,Z 609.607,A -85,B 0,C 180,E1 12855.046,E2 12855.046} C_VEL
LIN {X 0,Y 234.33,Z 603.345,A -85,B 0,C 180,E1 12850.303,E2 12850.303} C_VEL
LIN {X 0,Y 237,Z 595.196,A -85,B 0,C 180,E1 12845.581,E2 12845.581} C_VEL
LIN {X 0,Y 240.725,Z 585.601,A -85,B 0,C 180,E1 12841.198,E2 12841.198} C_VEL
LIN {X 0,Y 245.611,Z 574.045,A -85,B 0,C 180,E1 12836.992,E2 12836.992} C_VEL
LIN {X 0,Y 251.075,Z 561.523,A -85,B 0,C 180,E1 12833.322,E2 12833.322} C_VEL
LIN {X 0,Y 257.406,Z 546.777,A -85,B 0,C 180,E1 12829.851,E2 12829.851} C_VEL
LIN {X 0,Y 263.921,Z 530.89,A -85,B 0,C 180,E1 12826.859,E2 12826.859} C_VEL
LIN {X 0,Y 270.366,Z 513.946,A -85,B 0,C 180,E1 12824.311,E2 12824.311} C_VEL
LIN {X 0,Y 276.515,Z 495.982,A -85,B 0,C 180,E1 12822.163,E2 12822.163} C_VEL
LIN {X 0,Y 281.909,Z 478.015,A -85,B 0,C 180,E1 12820.47,E2 12820.47} C_VEL
LIN {X 0,Y 286.674,Z 459.427,A -85,B 0,C 180,E1 12819.104,E2 12819.104} C_VEL
LIN {X 0,Y 290.899,Z 439.071,A -85,B 0,C 180,E1 12817.983,E2 12817.983} C_VEL
LIN {X 0,Y 294.111,Z 417.748,A -85,B 0,C 180,E1 12817.152,E2 12817.152} C_VEL
LIN {X 0,Y 296.437,Z 390.018,A -85,B 0,C 180,E1 12816.422,E2 12816.422} C_VEL
LIN {X 0,Y 306.325,Z 246.061,A -85,B 0,C 180,E1 12813.06,E2 12813.06} C_VEL
LIN {X 0,Y 298.592,Z 231.672,A -85,B 0,C 180,E1 12810.317,E2 12810.317} C_VEL
LIN {X 0,Y 291.912,Z 220.468,A -85,B 0,C 180,E1 12807.708,E2 12807.708} C_VEL
LIN {X 0,Y 284.595,Z 209.105,A -85,B 0,C 180,E1 12804.491,E2 12804.491} C_VEL
LIN {X 0,Y 278.496,Z 200.542,A -85,B 0,C 180,E1 12801.426,E2 12801.426} C_VEL
LIN {X 0,Y 274.998,Z 195.722,A -85,B 0,C 180,E1 12799.431,E2 12799.431} C_VEL
LIN {X 0,Y 270.811,Z 190.251,A -85,B 0,C 180,E1 12796.737,E2 12796.737} C_VEL
LIN {X 0,Y 267.768,Z 186.442,A -85,B 0,C 180,E1 12794.488,E2 12794.488} C_VEL
LIN {X 0,Y 263.802,Z 181.39,A -85,B 0,C 180,E1 12790.924,E2 12790.924} C_VEL
LIN {X 0,Y 259.592,Z 176.309,A -85,B 0,C 180,E1 12785.525,E2 12785.525} C_VEL
LIN {X 0,Y 258.65,Z 175.392,A -85,B 0,C 180,E1 12783.768,E2 12783.768} C_VEL
LIN {X 0,Y 257.067,Z 174.303,A -85,B 0,C 180,E1 12777.993,E2 12777.993} C_VEL
LIN {X 0,Y 257.878,Z 175.035,A -85,B 0,C 180,E1 12772.2,E2 12772.2} C_VEL
LIN {X 0,Y 258.807,Z 175.979,A -85,B 0,C 180,E1 12769.988,E2 12769.988} C_VEL
LIN {X 0,Y 263.092,Z 181.584,A -85,B 0,C 180,E1 12763.893,E2 12763.893} C_VEL
LIN {X 0,Y 267.178,Z 186.83,A -85,B 0,C 180,E1 12760.089,E2 12760.089} C_VEL
LIN {X 0,Y 271.484,Z 192.576,A -85,B 0,C 180,E1 12756.906,E2 12756.906} C_VEL
LIN {X 0,Y 277.347,Z 200.667,A -85,B 0,C 180,E1 12753.331,E2 12753.331} C_VEL
LIN {X 0,Y 283.178,Z 209.259,A -85,B 0,C 180,E1 12750.316,E2 12750.316} C_VEL
LIN {X 0,Y 289.855,Z 219.789,A -85,B 0,C 180,E1 12747.308,E2 12747.308} C_VEL
LIN {X 0,Y 296.816,Z 231.718,A -85,B 0,C 180,E1 12744.532,E2 12744.532} C_VEL
LIN {X 0,Y 303.989,Z 245.209,A -85,B 0,C 180,E1 12741.953,E2 12741.953} C_VEL
LIN {X 0,Y 305.27,Z 248.291,A -85,B 0,C 180,E1 12741.497,E2 12741.497} C_VEL
LIN {X 0,Y 295.927,Z 398.793,A -85,B 0,C 180,E1 12738.23,E2 12738.23} C_VEL
LIN {X 0,Y 293.53,Z 418.545,A -85,B 0,C 180,E1 12737.505,E2 12737.505} C_VEL
LIN {X 0,Y 290.177,Z 437.453,A -85,B 0,C 180,E1 12736.493,E2 12736.493} C_VEL
LIN {X 0,Y 286.028,Z 455.337,A -85,B 0,C 180,E1 12735.202,E2 12735.202} C_VEL
LIN {X 0,Y 280.912,Z 473.199,A -85,B 0,C 180,E1 12733.528,E2 12733.528} C_VEL
LIN {X 0,Y 275.234,Z 489.907,A -85,B 0,C 180,E1 12731.525,E2 12731.525} C_VEL
LIN {X 0,Y 269.149,Z 505.511,A -85,B 0,C 180,E1 12729.161,E2 12729.161} C_VEL
LIN {X 0,Y 262.828,Z 519.997,A -85,B 0,C 180,E1 12726.401,E2 12726.401} C_VEL
LIN {X 0,Y 256.689,Z 532.892,A -85,B 0,C 180,E1 12723.312,E2 12723.312} C_VEL
LIN {X 0,Y 250.57,Z 544.951,A -85,B 0,C 180,E1 12719.655,E2 12719.655} C_VEL
LIN {X 0,Y 245.101,Z 555.293,A -85,B 0,C 180,E1 12715.619,E2 12715.619} C_VEL
LIN {X 0,Y 240.718,Z 563.563,A -85,B 0,C 180,E1 12711.438,E2 12711.438} C_VEL
LIN {X 0,Y 237.242,Z 570.315,A -85,B 0,C 180,E1 12706.904,E2 12706.904} C_VEL
LIN {X 0,Y 234.807,Z 575.453,A -85,B 0,C 180,E1 12702.042,E2 12702.042} C_VEL
LIN {X 0,Y 233.448,Z 578.758,A -85,B 0,C 180,E1 12697.133,E2 12697.133} C_VEL
LIN {X 0,Y 232.923,Z 580.323,A -85,B 0,C 180,E1 12692.459,E2 12692.459} C_VEL
LIN {X 0,Y 232.906,Z 580.362,A -85,B 0,C 180,E1 12687.784,E2 12687.784} C_VEL
LIN {X 0,Y 233.388,Z 578.919,A -85,B 0,C 180,E1 12683.109,E2 12683.109} C_VEL
LIN {X 0,Y 234.599,Z 575.936,A -85,B 0,C 180,E1 12678.443,E2 12678.443} C_VEL
LIN {X 0,Y 236.753,Z 571.312,A -85,B 0,C 180,E1 12673.814,E2 12673.814} C_VEL
LIN {X 0,Y 240.027,Z 564.908,A -85,B 0,C 180,E1 12669.262,E2 12669.262} C_VEL
LIN {X 0,Y 244.213,Z 557.016,A -85,B 0,C 180,E1 12665.056,E2 12665.056} C_VEL
LIN {X 0,Y 249.485,Z 547.089,A -85,B 0,C 180,E1 12660.991,E2 12660.991} C_VEL
LIN {X 0,Y 255.056,Z 536.263,A -85,B 0,C 180,E1 12657.515,E2 12657.515} C_VEL
LIN {X 0,Y 261.422,Z 523.152,A -85,B 0,C 180,E1 12654.183,E2 12654.183} C_VEL
LIN {X 0,Y 267.62,Z 509.307,A -85,B 0,C 180,E1 12651.395,E2 12651.395} C_VEL
LIN {X 0,Y 273.849,Z 493.83,A -85,B 0,C 180,E1 12648.912,E2 12648.912} C_VEL
LIN {X 0,Y 279.714,Z 477.186,A -85,B 0,C 180,E1 12646.8,E2 12646.8} C_VEL
LIN {X 0,Y 284.792,Z 460.303,A -85,B 0,C 180,E1 12645.114,E2 12645.114} C_VEL
LIN {X 0,Y 289.197,Z 442.505,A -85,B 0,C 180,E1 12643.73,E2 12643.73} C_VEL
LIN {X 0,Y 292.834,Z 423.557,A -85,B 0,C 180,E1 12642.623,E2 12642.623} C_VEL
LIN {X 0,Y 295.507,Z 403.959,A -85,B 0,C 180,E1 12641.822,E2 12641.822} C_VEL
LIN {X 0,Y 295.687,Z 401.762,A -85,B 0,C 180,E1 12641.739,E2 12641.739} C_VEL
LIN {X 0,Y 291.445,Z 408.925,A -85,B 0,C 180,E1 12641.136,E2 12641.136} C_VEL
LIN {X 0,Y 290.331,Z 410.828,A -85,B 0,C 180,E1 12641,E2 12641} C_VEL
LIN {X 0,Y 290.117,Z 411.398,A -85,B 0,C 180,E1 12640.99,E2 12640.99} C_VEL
LIN {X 0,Y 282.472,Z 430.226,A -85,B 0,C 180,E1 12640.687,E2 12640.687} C_VEL
LIN {X 0,Y 276.85,Z 440.41,A -85,B 0,C 180,E1 12640.381,E2 12640.381} C_VEL
LIN {X 0,Y 275.685,Z 442.15,A -85,B 0,C 180,E1 12640.297,E2 12640.297} C_VEL
LIN {X 0,Y 270.45,Z 448.852,A -85,B 0,C 180,E1 12639.761,E2 12639.761} C_VEL
LIN {X 0,Y 265.325,Z 453.478,A -85,B 0,C 180,E1 12639.001,E2 12639.001} C_VEL
LIN {X 0,Y 261.861,Z 455.94,A -85,B 0,C 180,E1 12638.351,E2 12638.351} C_VEL
LIN {X 0,Y 256.825,Z 460.986,A -85,B 0,C 180,E1 12637.679,E2 12637.679} C_VEL
LIN {X 0,Y 252.997,Z 463.591,A -85,B 0,C 180,E1 12636.922,E2 12636.922} C_VEL
LIN {X 0,Y 250.854,Z 464.538,A -85,B 0,C 180,E1 12636.375,E2 12636.375} C_VEL
LIN {X 0,Y 246.654,Z 468.445,A -85,B 0,C 180,E1 12635.714,E2 12635.714} C_VEL
LIN {X 0,Y 243.836,Z 469.996,A -85,B 0,C 180,E1 12635.036,E2 12635.036} C_VEL
LIN {X 0,Y 242.166,Z 470.087,A -85,B 0,C 180,E1 12634.332,E2 12634.332} C_VEL
LIN {X 0,Y 238.939,Z 488.335,A -85,B 0,C 180,E1 12631.821,E2 12631.821} C_VEL
LIN {X 0,Y 235.706,Z 505.342,A -85,B 0,C 180,E1 12628.92,E2 12628.92} C_VEL
LIN {X 0,Y 232.709,Z 520.692,A -85,B 0,C 180,E1 12625.72,E2 12625.72} C_VEL
LIN {X 0,Y 230.064,Z 534.489,A -85,B 0,C 180,E1 12622.217,E2 12622.217} C_VEL
LIN {X 0,Y 227.893,Z 546.684,A -85,B 0,C 180,E1 12618.415,E2 12618.415} C_VEL
LIN {X 0,Y 226.347,Z 556.74,A -85,B 0,C 180,E1 12614.584,E2 12614.584} C_VEL
LIN {X 0,Y 225.318,Z 565.39,A -85,B 0,C 180,E1 12610.483,E2 12610.483} C_VEL
LIN {X 0,Y 224.812,Z 572.24,A -85,B 0,C 180,E1 12606.384,E2 12606.384} C_VEL
LIN {X 0,Y 224.712,Z 577.486,A -85,B 0,C 180,E1 12602.296,E2 12602.296} C_VEL
LIN {X 0,Y 224.974,Z 581.408,A -85,B 0,C 180,E1 12597.963,E2 12597.963} C_VEL
LIN {X 0,Y 225.786,Z 583.877,A -85,B 0,C 180,E1 12593.389,E2 12593.389} C_VEL
LIN {X 0,Y 227.406,Z 584.715,A -85,B 0,C 180,E1 12588.846,E2 12588.846} C_VEL
LIN {X 0,Y 230.21,Z 583.873,A -85,B 0,C 180,E1 12584.12,E2 12584.12} C_VEL
LIN {X 0,Y 234.563,Z 581.137,A -85,B 0,C 180,E1 12579.281,E2 12579.281} C_VEL
LIN {X 0,Y 240.432,Z 576.511,A -85,B 0,C 180,E1 12574.639,E2 12574.639} C_VEL
LIN {X 0,Y 247.847,Z 570.014,A -85,B 0,C 180,E1 12570.251,E2 12570.251} C_VEL
LIN {X 0,Y 256.774,Z 561.529,A -85,B 0,C 180,E1 12566.164,E2 12566.164} C_VEL
LIN {X 0,Y 267.789,Z 550.575,A -85,B 0,C 180,E1 12562.242,E2 12562.242} C_VEL
LIN {X 0,Y 279.196,Z 538.771,A -85,B 0,C 180,E1 12559.054,E2 12559.054} C_VEL
LIN {X 0,Y 281.621,Z 536.148,A -85,B 0,C 180,E1 12558.41,E2 12558.41} C_VEL
LIN {X 0,Y 266.599,Z 552.23,A -85,B 0,C 180,E1 12554.837,E2 12554.837} C_VEL
LIN {X 0,Y 254.236,Z 566.327,A -85,B 0,C 180,E1 12550.758,E2 12550.758} C_VEL
LIN {X 0,Y 243.247,Z 580.035,A -85,B 0,C 180,E1 12545.712,E2 12545.712} C_VEL
LIN {X 0,Y 235.083,Z 591.451,A -85,B 0,C 180,E1 12540.3,E2 12540.3} C_VEL
LIN {X 0,Y 229.713,Z 600.163,A -85,B 0,C 180,E1 12534.976,E2 12534.976} C_VEL
LIN {X 0,Y 226.367,Z 606.82,A -85,B 0,C 180,E1 12529.616,E2 12529.616} C_VEL
LIN {X 0,Y 224.737,Z 611.404,A -85,B 0,C 180,E1 12524.429,E2 12524.429} C_VEL
LIN {X 0,Y 224.381,Z 615.515,A -85,B 0,C 180,E1 12517.426,E2 12517.426} C_VEL
LIN {X 0,Y 224.594,Z 617.198,A -85,B 0,C 180,E1 12513.064,E2 12513.064} C_VEL
LIN {X 0,Y 224.675,Z 617.465,A -85,B 0,C 180,E1 12508.982,E2 12508.982} C_VEL
LIN {X 0,Y 224.49,Z 616.572,A -85,B 0,C 180,E1 12504.891,E2 12504.891} C_VEL
LIN {X 0,Y 224.35,Z 614.063,A -85,B 0,C 180,E1 12500.251,E2 12500.251} C_VEL
LIN {X 0,Y 224.793,Z 609.804,A -85,B 0,C 180,E1 12495.315,E2 12495.315} C_VEL
LIN {X 0,Y 226.255,Z 603.815,A -85,B 0,C 180,E1 12490.377,E2 12490.377} C_VEL
LIN {X 0,Y 228.952,Z 595.981,A -85,B 0,C 180,E1 12485.49,E2 12485.49} C_VEL
LIN {X 0,Y 232.995,Z 586.112,A -85,B 0,C 180,E1 12480.713,E2 12480.713} C_VEL
LIN {X 0,Y 238.121,Z 574.649,A -85,B 0,C 180,E1 12476.342,E2 12476.342} C_VEL
LIN {X 0,Y 244.105,Z 561.622,A -85,B 0,C 180,E1 12472.391,E2 12472.391} C_VEL
LIN {X 0,Y 250.423,Z 547.629,A -85,B 0,C 180,E1 12468.991,E2 12468.991} C_VEL
LIN {X 0,Y 256.884,Z 532.653,A -85,B 0,C 180,E1 12466.059,E2 12466.059} C_VEL
LIN {X 0,Y 263.367,Z 516.554,A -85,B 0,C 180,E1 12463.523,E2 12463.523} C_VEL
LIN {X 0,Y 269.665,Z 499.24,A -85,B 0,C 180,E1 12461.341,E2 12461.341} C_VEL
LIN {X 0,Y 275.472,Z 481.153,A -85,B 0,C 180,E1 12459.54,E2 12459.54} C_VEL
LIN {X 0,Y 280.677,Z 462.164,A -85,B 0,C 180,E1 12458.071,E2 12458.071} C_VEL
LIN {X 0,Y 285.068,Z 442.583,A -85,B 0,C 180,E1 12456.933,E2 12456.933} C_VEL
LIN {X 0,Y 288.503,Z 422.162,A -85,B 0,C 180,E1 12456.076,E2 12456.076} C_VEL
LIN {X 0,Y 290.715,Z 400.556,A -85,B 0,C 180,E1 12455.449,E2 12455.449} C_VEL
LIN {X 0,Y 301.446,Z 249.659,A -85,B 0,C 180,E1 12451.912,E2 12451.912} C_VEL
LIN {X 0,Y 294.197,Z 236.053,A -85,B 0,C 180,E1 12449.189,E2 12449.189} C_VEL
LIN {X 0,Y 287.661,Z 224.905,A -85,B 0,C 180,E1 12446.472,E2 12446.472} C_VEL
LIN {X 0,Y 280.099,Z 213.13,A -85,B 0,C 180,E1 12442.898,E2 12442.898} C_VEL
LIN {X 0,Y 273.664,Z 203.819,A -85,B 0,C 180,E1 12439.308,E2 12439.308} C_VEL
LIN {X 0,Y 268.793,Z 197.433,A -85,B 0,C 180,E1 12436.088,E2 12436.088} C_VEL
LIN {X 0,Y 265.99,Z 193.855,A -85,B 0,C 180,E1 12433.92,E2 12433.92} C_VEL
LIN {X 0,Y 262.331,Z 189.055,A -85,B 0,C 180,E1 12430.479,E2 12430.479} C_VEL
LIN {X 0,Y 258.012,Z 183.54,A -85,B 0,C 180,E1 12424.445,E2 12424.445} C_VEL
LIN {X 0,Y 256.099,Z 182.244,A -85,B 0,C 180,E1 12418.086,E2 12418.086} C_VEL
LIN {X 0,Y 256.834,Z 182.93,A -85,B 0,C 180,E1 12412.393,E2 12412.393} C_VEL
LIN {X 0,Y 257.729,Z 183.881,A -85,B 0,C 180,E1 12410.171,E2 12410.171} C_VEL
LIN {X 0,Y 261.734,Z 189.303,A -85,B 0,C 180,E1 12404.262,E2 12404.262} C_VEL
LIN {X 0,Y 265.587,Z 194.415,A -85,B 0,C 180,E1 12400.538,E2 12400.538} C_VEL
LIN {X 0,Y 269.701,Z 200.08,A -85,B 0,C 180,E1 12397.381,E2 12397.381} C_VEL
LIN {X 0,Y 275.175,Z 207.856,A -85,B 0,C 180,E1 12393.917,E2 12393.917} C_VEL
LIN {X 0,Y 280.669,Z 216.165,A -85,B 0,C 180,E1 12390.962,E2 12390.962} C_VEL
LIN {X 0,Y 287.045,Z 226.518,A -85,B 0,C 180,E1 12387.972,E2 12387.972} C_VEL
LIN {X 0,Y 293.875,Z 238.537,A -85,B 0,C 180,E1 12385.138,E2 12385.138} C_VEL
LIN {X 0,Y 300.455,Z 251.472,A -85,B 0,C 180,E1 12382.669,E2 12382.669} C_VEL
LIN {X 0,Y 290.907,Z 399.085,A -85,B 0,C 180,E1 12379.446,E2 12379.446} C_VEL
LIN {X 0,Y 288.425,Z 418.852,A -85,B 0,C 180,E1 12378.718,E2 12378.718} C_VEL
LIN {X 0,Y 285.068,Z 437.257,A -85,B 0,C 180,E1 12377.735,E2 12377.735} C_VEL
LIN {X 0,Y 280.7,Z 455.531,A -85,B 0,C 180,E1 12376.418,E2 12376.418} C_VEL
LIN {X 0,Y 275.471,Z 473.217,A -85,B 0,C 180,E1 12374.759,E2 12374.759} C_VEL
LIN {X 0,Y 269.581,Z 490.008,A -85,B 0,C 180,E1 12372.743,E2 12372.743} C_VEL
LIN {X 0,Y 263.251,Z 505.682,A -85,B 0,C 180,E1 12370.357,E2 12370.357} C_VEL
LIN {X 0,Y 256.886,Z 519.741,A -85,B 0,C 180,E1 12367.665,E2 12367.665} C_VEL
LIN {X 0,Y 250.437,Z 532.775,A -85,B 0,C 180,E1 12364.534,E2 12364.534} C_VEL
LIN {X 0,Y 244.335,Z 544.302,A -85,B 0,C 180,E1 12361.036,E2 12361.036} C_VEL
LIN {X 0,Y 238.765,Z 554.366,A -85,B 0,C 180,E1 12357.156,E2 12357.156} C_VEL
LIN {X 0,Y 233.951,Z 562.946,A -85,B 0,C 180,E1 12352.885,E2 12352.885} C_VEL
LIN {X 0,Y 230.073,Z 569.999,A -85,B 0,C 180,E1 12348.232,E2 12348.232} C_VEL
LIN {X 0,Y 227.392,Z 575.201,A -85,B 0,C 180,E1 12343.475,E2 12343.475} C_VEL
LIN {X 0,Y 225.786,Z 578.712,A -85,B 0,C 180,E1 12338.658,E2 12338.658} C_VEL
LIN {X 0,Y 225.032,Z 580.658,A -85,B 0,C 180,E1 12333.82,E2 12333.82} C_VEL
LIN {X 0,Y 224.891,Z 581.109,A -85,B 0,C 180,E1 12328.979,E2 12328.979} C_VEL
LIN {X 0,Y 225.252,Z 580.089,A -85,B 0,C 180,E1 12324.139,E2 12324.139} C_VEL
LIN {X 0,Y 226.325,Z 577.548,A -85,B 0,C 180,E1 12319.305,E2 12319.305} C_VEL
LIN {X 0,Y 228.421,Z 573.231,A -85,B 0,C 180,E1 12314.367,E2 12314.367} C_VEL
LIN {X 0,Y 231.704,Z 567.098,A -85,B 0,C 180,E1 12309.54,E2 12309.54} C_VEL
LIN {X 0,Y 236.077,Z 559.273,A -85,B 0,C 180,E1 12305.008,E2 12305.008} C_VEL
LIN {X 0,Y 241.177,Z 550.2,A -85,B 0,C 180,E1 12300.983,E2 12300.983} C_VEL
LIN {X 0,Y 247.183,Z 539.178,A -85,B 0,C 180,E1 12297.176,E2 12297.176} C_VEL
LIN {X 0,Y 253.678,Z 526.551,A -85,B 0,C 180,E1 12293.755,E2 12293.755} C_VEL
LIN {X 0,Y 260.237,Z 512.746,A -85,B 0,C 180,E1 12290.799,E2 12290.799} C_VEL
LIN {X 0,Y 266.614,Z 497.9,A -85,B 0,C 180,E1 12288.271,E2 12288.271} C_VEL
LIN {X 0,Y 272.625,Z 482.014,A -85,B 0,C 180,E1 12286.117,E2 12286.117} C_VEL
LIN {X 0,Y 278.109,Z 465.185,A -85,B 0,C 180,E1 12284.319,E2 12284.319} C_VEL
LIN {X 0,Y 282.922,Z 447.357,A -85,B 0,C 180,E1 12282.833,E2 12282.833} C_VEL
LIN {X 0,Y 286.715,Z 429.32,A -85,B 0,C 180,E1 12281.679,E2 12281.679} C_VEL
LIN {X 0,Y 281.838,Z 435.898,A -85,B 0,C 180,E1 12281.155,E2 12281.155} C_VEL
LIN {X 0,Y 277.175,Z 440.556,A -85,B 0,C 180,E1 12280.491,E2 12280.491} C_VEL
LIN {X 0,Y 275.875,Z 441.873,A -85,B 0,C 180,E1 12280.312,E2 12280.312} C_VEL
LIN {X 0,Y 275.685,Z 442.15,A -85,B 0,C 180,E1 12280.297,E2 12280.297} C_VEL
LIN {X 0,Y 270.555,Z 450.435,A -85,B 0,C 180,E1 12280.037,E2 12280.037} C_VEL
LIN {X 0,Y 264.796,Z 459.149,A -85,B 0,C 180,E1 12279.792,E2 12279.792} C_VEL
LIN {X 0,Y 262.43,Z 461.885,A -85,B 0,C 180,E1 12279.597,E2 12279.597} C_VEL
LIN {X 0,Y 256.707,Z 467.119,A -85,B 0,C 180,E1 12278.836,E2 12278.836} C_VEL
LIN {X 0,Y 251.978,Z 470.086,A -85,B 0,C 180,E1 12277.956,E2 12277.956} C_VEL
LIN {X 0,Y 250.528,Z 470.819,A -85,B 0,C 180,E1 12277.635,E2 12277.635} C_VEL
LIN {X 0,Y 246.163,Z 474.395,A -85,B 0,C 180,E1 12276.952,E2 12276.952} C_VEL
LIN {X 0,Y 242.504,Z 476.47,A -85,B 0,C 180,E1 12276.129,E2 12276.129} C_VEL
LIN {X 0,Y 240.594,Z 477.11,A -85,B 0,C 180,E1 12275.579,E2 12275.579} C_VEL
LIN {X 0,Y 236.391,Z 480.258,A -85,B 0,C 180,E1 12274.821,E2 12274.821} C_VEL
LIN {X 0,Y 233.813,Z 481.298,A -85,B 0,C 180,E1 12274.07,E2 12274.07} C_VEL
LIN {X 0,Y 232.631,Z 481.16,A -85,B 0,C 180,E1 12273.47,E2 12273.47} C_VEL
LIN {X 0,Y 229.306,Z 498.627,A -85,B 0,C 180,E1 12270.675,E2 12270.675} C_VEL
LIN {X 0,Y 226.109,Z 514.682,A -85,B 0,C 180,E1 12267.523,E2 12267.523} C_VEL
LIN {X 0,Y 223.231,Z 529.16,A -85,B 0,C 180,E1 12264.054,E2 12264.054} C_VEL
LIN {X 0,Y 220.714,Z 542.364,A -85,B 0,C 180,E1 12260.139,E2 12260.139} C_VEL
LIN {X 0,Y 218.879,Z 553.284,A -85,B 0,C 180,E1 12256.18,E2 12256.18} C_VEL
LIN {X 0,Y 217.579,Z 563.05,A -85,B 0,C 180,E1 12251.807,E2 12251.807} C_VEL
LIN {X 0,Y 216.896,Z 570.823,A -85,B 0,C 180,E1 12247.417,E2 12247.417} C_VEL
LIN {X 0,Y 216.708,Z 576.911,A -85,B 0,C 180,E1 12242.91,E2 12242.91} C_VEL
LIN {X 0,Y 216.932,Z 581.287,A -85,B 0,C 180,E1 12238.416,E2 12238.416} C_VEL
LIN {X 0,Y 217.716,Z 584.235,A -85,B 0,C 180,E1 12233.673,E2 12233.673} C_VEL
LIN {X 0,Y 219.344,Z 585.552,A -85,B 0,C 180,E1 12228.963,E2 12228.963} C_VEL
LIN {X 0,Y 222.214,Z 585.253,A -85,B 0,C 180,E1 12224.07,E2 12224.07} C_VEL
LIN {X 0,Y 226.71,Z 583.128,A -85,B 0,C 180,E1 12219.07,E2 12219.07} C_VEL
LIN {X 0,Y 232.787,Z 579.137,A -85,B 0,C 180,E1 12214.291,E2 12214.291} C_VEL
LIN {X 0,Y 240.455,Z 573.308,A -85,B 0,C 180,E1 12209.792,E2 12209.792} C_VEL
LIN {X 0,Y 250.537,Z 564.98,A -85,B 0,C 180,E1 12205.299,E2 12205.299} C_VEL
LIN {X 0,Y 261.659,Z 555.222,A -85,B 0,C 180,E1 12201.475,E2 12201.475} C_VEL
LIN {X 0,Y 272.314,Z 545.459,A -85,B 0,C 180,E1 12198.508,E2 12198.508} C_VEL
LIN {X 0,Y 257.761,Z 559.542,A -85,B 0,C 180,E1 12194.91,E2 12194.91} C_VEL
LIN {X 0,Y 244.919,Z 572.84,A -85,B 0,C 180,E1 12190.476,E2 12190.476} C_VEL
LIN {X 0,Y 234.023,Z 585.1,A -85,B 0,C 180,E1 12185.226,E2 12185.226} C_VEL
LIN {X 0,Y 225.859,Z 595.436,A -85,B 0,C 180,E1 12179.433,E2 12179.433} C_VEL
LIN {X 0,Y 220.707,Z 603.112,A -85,B 0,C 180,E1 12173.78,E2 12173.78} C_VEL
LIN {X 0,Y 217.649,Z 608.884,A -85,B 0,C 180,E1 12167.928,E2 12167.928} C_VEL
LIN {X 0,Y 216.457,Z 612.482,A -85,B 0,C 180,E1 12162.27,E2 12162.27} C_VEL
LIN {X 0,Y 216.463,Z 615.755,A -85,B 0,C 180,E1 12155.834,E2 12155.834} C_VEL
LIN {X 0,Y 216.681,Z 616.771,A -85,B 0,C 180,E1 12151.588,E2 12151.588} C_VEL
LIN {X 0,Y 216.648,Z 616.686,A -85,B 0,C 180,E1 12147.621,E2 12147.621} C_VEL
LIN {X 0,Y 216.418,Z 615.233,A -85,B 0,C 180,E1 12143.103,E2 12143.103} C_VEL
LIN {X 0,Y 216.434,Z 612.281,A -85,B 0,C 180,E1 12138.274,E2 12138.274} C_VEL
LIN {X 0,Y 217.278,Z 607.466,A -85,B 0,C 180,E1 12133.149,E2 12133.149} C_VEL
LIN {X 0,Y 219.293,Z 600.849,A -85,B 0,C 180,E1 12128.047,E2 12128.047} C_VEL
LIN {X 0,Y 222.456,Z 592.846,A -85,B 0,C 180,E1 12123.293,E2 12123.293} C_VEL
LIN {X 0,Y 226.911,Z 582.995,A -85,B 0,C 180,E1 12118.673,E2 12118.673} C_VEL
LIN {X 0,Y 232.657,Z 571.021,A -85,B 0,C 180,E1 12114.237,E2 12114.237} C_VEL
LIN {X 0,Y 238.834,Z 558.303,A -85,B 0,C 180,E1 12110.483,E2 12110.483} C_VEL
LIN {X 0,Y 245.494,Z 544.223,A -85,B 0,C 180,E1 12107.146,E2 12107.146} C_VEL
LIN {X 0,Y 252.444,Z 528.665,A -85,B 0,C 180,E1 12104.193,E2 12104.193} C_VEL
LIN {X 0,Y 259.454,Z 511.575,A -85,B 0,C 180,E1 12101.618,E2 12101.618} C_VEL
LIN {X 0,Y 266.125,Z 493.353,A -85,B 0,C 180,E1 12099.461,E2 12099.461} C_VEL
LIN {X 0,Y 271.935,Z 475.028,A -85,B 0,C 180,E1 12097.769,E2 12097.769} C_VEL
LIN {X 0,Y 277.037,Z 455.854,A -85,B 0,C 180,E1 12096.409,E2 12096.409} C_VEL
LIN {X 0,Y 281.259,Z 435.981,A -85,B 0,C 180,E1 12095.363,E2 12095.363} C_VEL
LIN {X 0,Y 284.383,Z 415.597,A -85,B 0,C 180,E1 12094.601,E2 12094.601} C_VEL
LIN {X 0,Y 286.96,Z 385.384,A -85,B 0,C 180,E1 12093.823,E2 12093.823} C_VEL
LIN {X 0,Y 296.659,Z 253.221,A -85,B 0,C 180,E1 12090.716,E2 12090.716} C_VEL
LIN {X 0,Y 290.029,Z 240.631,A -85,B 0,C 180,E1 12088.071,E2 12088.071} C_VEL
LIN {X 0,Y 283.527,Z 229.531,A -85,B 0,C 180,E1 12085.202,E2 12085.202} C_VEL
LIN {X 0,Y 277.397,Z 219.75,A -85,B 0,C 180,E1 12082.127,E2 12082.127} C_VEL
LIN {X 0,Y 271.51,Z 210.974,A -85,B 0,C 180,E1 12078.686,E2 12078.686} C_VEL
LIN {X 0,Y 266.946,Z 204.789,A -85,B 0,C 180,E1 12075.533,E2 12075.533} C_VEL
LIN {X 0,Y 264.367,Z 201.395,A -85,B 0,C 180,E1 12073.45,E2 12073.45} C_VEL
LIN {X 0,Y 260.99,Z 196.811,A -85,B 0,C 180,E1 12070.15,E2 12070.15} C_VEL
LIN {X 0,Y 256.912,Z 191.427,A -85,B 0,C 180,E1 12064.24,E2 12064.24} C_VEL
LIN {X 0,Y 255.112,Z 190.183,A -85,B 0,C 180,E1 12057.978,E2 12057.978} C_VEL
LIN {X 0,Y 255.865,Z 190.891,A -85,B 0,C 180,E1 12052.364,E2 12052.364} C_VEL
LIN {X 0,Y 256.656,Z 191.785,A -85,B 0,C 180,E1 12050.356,E2 12050.356} C_VEL
LIN {X 0,Y 260.387,Z 197.021,A -85,B 0,C 180,E1 12044.635,E2 12044.635} C_VEL
LIN {X 0,Y 263.956,Z 201.897,A -85,B 0,C 180,E1 12041.045,E2 12041.045} C_VEL
LIN {X 0,Y 267.877,Z 207.476,A -85,B 0,C 180,E1 12037.91,E2 12037.91} C_VEL
LIN {X 0,Y 273.035,Z 215.037,A -85,B 0,C 180,E1 12034.514,E2 12034.514} C_VEL
LIN {X 0,Y 278.471,Z 223.524,A -85,B 0,C 180,E1 12031.475,E2 12031.475} C_VEL
LIN {X 0,Y 284.403,Z 233.473,A -85,B 0,C 180,E1 12028.587,E2 12028.587} C_VEL
LIN {X 0,Y 290.972,Z 245.376,A -85,B 0,C 180,E1 12025.757,E2 12025.757} C_VEL
LIN {X 0,Y 295.745,Z 255.09,A -85,B 0,C 180,E1 12023.869,E2 12023.869} C_VEL
LIN {X 0,Y 286.016,Z 399.426,A -85,B 0,C 180,E1 12020.702,E2 12020.702} C_VEL
LIN {X 0,Y 283.435,Z 419.268,A -85,B 0,C 180,E1 12019.969,E2 12019.969} C_VEL
LIN {X 0,Y 279.798,Z 438.407,A -85,B 0,C 180,E1 12018.937,E2 12018.937} C_VEL
LIN {X 0,Y 275.259,Z 456.631,A -85,B 0,C 180,E1 12017.606,E2 12017.606} C_VEL
LIN {X 0,Y 269.884,Z 474.106,A -85,B 0,C 180,E1 12015.947,E2 12015.947} C_VEL
LIN {X 0,Y 263.786,Z 490.82,A -85,B 0,C 180,E1 12013.917,E2 12013.917} C_VEL
LIN {X 0,Y 256.968,Z 507.008,A -85,B 0,C 180,E1 12011.41,E2 12011.41} C_VEL
LIN {X 0,Y 250.138,Z 521.426,A -85,B 0,C 180,E1 12008.575,E2 12008.575} C_VEL
LIN {X 0,Y 243.463,Z 534.283,A -85,B 0,C 180,E1 12005.382,E2 12005.382} C_VEL
LIN {X 0,Y 237.133,Z 545.659,A -85,B 0,C 180,E1 12001.805,E2 12001.805} C_VEL
LIN {X 0,Y 231.037,Z 556.123,A -85,B 0,C 180,E1 11997.583,E2 11997.583} C_VEL
LIN {X 0,Y 225.893,Z 564.801,A -85,B 0,C 180,E1 11992.976,E2 11992.976} C_VEL
LIN {X 0,Y 221.896,Z 571.681,A -85,B 0,C 180,E1 11988.053,E2 11988.053} C_VEL
LIN {X 0,Y 219.157,Z 576.751,A -85,B 0,C 180,E1 11982.916,E2 11982.916} C_VEL
LIN {X 0,Y 217.648,Z 579.945,A -85,B 0,C 180,E1 11977.92,E2 11977.92} C_VEL
LIN {X 0,Y 216.985,Z 581.614,A -85,B 0,C 180,E1 11972.639,E2 11972.639} C_VEL
LIN {X 0,Y 216.966,Z 581.652,A -85,B 0,C 180,E1 11967.621,E2 11967.621} C_VEL
LIN {X 0,Y 217.526,Z 580.211,A -85,B 0,C 180,E1 11962.604,E2 11962.604} C_VEL
LIN {X 0,Y 218.921,Z 577.233,A -85,B 0,C 180,E1 11957.603,E2 11957.603} C_VEL
LIN {X 0,Y 221.383,Z 572.614,A -85,B 0,C 180,E1 11952.656,E2 11952.656} C_VEL
LIN {X 0,Y 225.078,Z 566.216,A -85,B 0,C 180,E1 11947.814,E2 11947.814} C_VEL
LIN {X 0,Y 229.75,Z 558.336,A -85,B 0,C 180,E1 11943.367,E2 11943.367} C_VEL
LIN {X 0,Y 235.581,Z 548.427,A -85,B 0,C 180,E1 11939.098,E2 11939.098} C_VEL
LIN {X 0,Y 242.101,Z 536.885,A -85,B 0,C 180,E1 11935.253,E2 11935.253} C_VEL
LIN {X 0,Y 248.647,Z 524.514,A -85,B 0,C 180,E1 11932.014,E2 11932.014} C_VEL
LIN {X 0,Y 255.332,Z 510.775,A -85,B 0,C 180,E1 11929.158,E2 11929.158} C_VEL
LIN {X 0,Y 262.04,Z 495.384,A -85,B 0,C 180,E1 11926.619,E2 11926.619} C_VEL
LIN {X 0,Y 268.365,Z 478.78,A -85,B 0,C 180,E1 11924.463,E2 11924.463} C_VEL
LIN {X 0,Y 274.054,Z 461.189,A -85,B 0,C 180,E1 11922.678,E2 11922.678} C_VEL
LIN {X 0,Y 277.84,Z 447.237,A -85,B 0,C 180,E1 11921.536,E2 11921.536} C_VEL
LIN {X 0,Y 272.031,Z 454.056,A -85,B 0,C 180,E1 11921.002,E2 11921.002} C_VEL
LIN {X 0,Y 266.311,Z 459.077,A -85,B 0,C 180,E1 11920.224,E2 11920.224} C_VEL
LIN {X 0,Y 262.638,Z 461.667,A -85,B 0,C 180,E1 11919.619,E2 11919.619} C_VEL
LIN {X 0,Y 262.43,Z 461.885,A -85,B 0,C 180,E1 11919.597,E2 11919.597} C_VEL
LIN {X 0,Y 247.795,Z 476.432,A -85,B 0,C 180,E1 11917.992,E2 11917.992} C_VEL
LIN {X 0,Y 239.366,Z 483.413,A -85,B 0,C 180,E1 11916.842,E2 11916.842} C_VEL
LIN {X 0,Y 238.604,Z 483.985,A -85,B 0,C 180,E1 11916.716,E2 11916.716} C_VEL
LIN {X 0,Y 234.064,Z 486.842,A -85,B 0,C 180,E1 11915.82,E2 11915.82} C_VEL
LIN {X 0,Y 230.195,Z 488.174,A -85,B 0,C 180,E1 11914.681,E2 11914.681} C_VEL
LIN {X 0,Y 226.248,Z 490.686,A -85,B 0,C 180,E1 11913.838,E2 11913.838} C_VEL
LIN {X 0,Y 223.9,Z 491.341,A -85,B 0,C 180,E1 11913.012,E2 11913.012} C_VEL
LIN {X 0,Y 223.105,Z 491.199,A -85,B 0,C 180,E1 11912.534,E2 11912.534} C_VEL
LIN {X 0,Y 219.715,Z 507.931,A -85,B 0,C 180,E1 11909.438,E2 11909.438} C_VEL
LIN {X 0,Y 216.594,Z 523.078,A -85,B 0,C 180,E1 11906.012,E2 11906.012} C_VEL
LIN {X 0,Y 213.837,Z 536.799,A -85,B 0,C 180,E1 11902.206,E2 11902.206} C_VEL
LIN {X 0,Y 211.657,Z 548.711,A -85,B 0,C 180,E1 11898.167,E2 11898.167} C_VEL
LIN {X 0,Y 210.05,Z 559.276,A -85,B 0,C 180,E1 11893.769,E2 11893.769} C_VEL
LIN {X 0,Y 209.123,Z 567.74,A -85,B 0,C 180,E1 11889.356,E2 11889.356} C_VEL
LIN {X 0,Y 208.734,Z 574.494,A -85,B 0,C 180,E1 11884.885,E2 11884.885} C_VEL
LIN {X 0,Y 208.795,Z 579.758,A -85,B 0,C 180,E1 11880.275,E2 11880.275} C_VEL
LIN {X 0,Y 209.358,Z 583.66,A -85,B 0,C 180,E1 11875.344,E2 11875.344} C_VEL
LIN {X 0,Y 210.71,Z 585.907,A -85,B 0,C 180,E1 11870.441,E2 11870.441} C_VEL
LIN {X 0,Y 213.29,Z 586.58,A -85,B 0,C 180,E1 11865.337,E2 11865.337} C_VEL
LIN {X 0,Y 217.515,Z 585.49,A -85,B 0,C 180,E1 11860.114,E2 11860.114} C_VEL
LIN {X 0,Y 223.389,Z 582.604,A -85,B 0,C 180,E1 11855.12,E2 11855.12} C_VEL
LIN {X 0,Y 231.335,Z 577.646,A -85,B 0,C 180,E1 11850.196,E2 11850.196} C_VEL
LIN {X 0,Y 241.077,Z 570.78,A -85,B 0,C 180,E1 11845.664,E2 11845.664} C_VEL
LIN {X 0,Y 252.562,Z 562.08,A -85,B 0,C 180,E1 11841.572,E2 11841.572} C_VEL
LIN {X 0,Y 262.874,Z 553.816,A -85,B 0,C 180,E1 11838.614,E2 11838.614} C_VEL
LIN {X 0,Y 249.466,Z 565.602,A -85,B 0,C 180,E1 11835.189,E2 11835.189} C_VEL
LIN {X 0,Y 235.478,Z 578.602,A -85,B 0,C 180,E1 11830.198,E2 11830.198} C_VEL
LIN {X 0,Y 224.745,Z 589.493,A -85,B 0,C 180,E1 11824.714,E2 11824.714} C_VEL
LIN {X 0,Y 216.805,Z 598.612,A -85,B 0,C 180,E1 11818.663,E2 11818.663} C_VEL
LIN {X 0,Y 211.761,Z 605.473,A -85,B 0,C 180,E1 11812.487,E2 11812.487} C_VEL
LIN {X 0,Y 209.224,Z 609.959,A -85,B 0,C 180,E1 11806.664,E2 11806.664} C_VEL
LIN {X 0,Y 208.367,Z 613.49,A -85,B 0,C 180,E1 11799.392,E2 11799.392} C_VEL
LIN {X 0,Y 208.553,Z 615.519,A -85,B 0,C 180,E1 11794.677,E2 11794.677} C_VEL
LIN {X 0,Y 208.736,Z 616.252,A -85,B 0,C 180,E1 11790.276,E2 11790.276} C_VEL
LIN {X 0,Y 208.584,Z 615.665,A -85,B 0,C 180,E1 11785.878,E2 11785.878} C_VEL
LIN {X 0,Y 208.373,Z 613.803,A -85,B 0,C 180,E1 11781.169,E2 11781.169} C_VEL
LIN {X 0,Y 208.693,Z 610.021,A -85,B 0,C 180,E1 11775.859,E2 11775.859} C_VEL
LIN {X 0,Y 210.103,Z 604.537,A -85,B 0,C 180,E1 11770.544,E2 11770.544} C_VEL
LIN {X 0,Y 212.846,Z 597.256,A -85,B 0,C 180,E1 11765.288,E2 11765.288} C_VEL
LIN {X 0,Y 217.053,Z 588.023,A -85,B 0,C 180,E1 11760.167,E2 11760.167} C_VEL
LIN {X 0,Y 222.433,Z 577.261,A -85,B 0,C 180,E1 11755.504,E2 11755.504} C_VEL
LIN {X 0,Y 228.721,Z 565.018,A -85,B 0,C 180,E1 11751.311,E2 11751.311} C_VEL
LIN {X 0,Y 235.718,Z 551.221,A -85,B 0,C 180,E1 11747.566,E2 11747.566} C_VEL
LIN {X 0,Y 242.594,Z 537.022,A -85,B 0,C 180,E1 11744.479,E2 11744.479} C_VEL
LIN {X 0,Y 250.087,Z 520.395,A -85,B 0,C 180,E1 11741.617,E2 11741.617} C_VEL
LIN {X 0,Y 257.346,Z 502.438,A -85,B 0,C 180,E1 11739.188,E2 11739.188} C_VEL
LIN {X 0,Y 263.82,Z 484.18,A -85,B 0,C 180,E1 11737.264,E2 11737.264} C_VEL
LIN {X 0,Y 269.633,Z 464.928,A -85,B 0,C 180,E1 11735.701,E2 11735.701} C_VEL
LIN {X 0,Y 274.322,Z 445.959,A -85,B 0,C 180,E1 11734.543,E2 11734.543} C_VEL
LIN {X 0,Y 278.133,Z 425.963,A -85,B 0,C 180,E1 11733.652,E2 11733.652} C_VEL
LIN {X 0,Y 280.711,Z 405.192,A -85,B 0,C 180,E1 11732.996,E2 11732.996} C_VEL
LIN {X 0,Y 292.063,Z 257.02,A -85,B 0,C 180,E1 11729.508,E2 11729.508} C_VEL
LIN {X 0,Y 285.963,Z 245.3,A -85,B 0,C 180,E1 11726.923,E2 11726.923} C_VEL
LIN {X 0,Y 279.456,Z 233.927,A -85,B 0,C 180,E1 11723.847,E2 11723.847} C_VEL
LIN {X 0,Y 273.79,Z 224.908,A -85,B 0,C 180,E1 11720.796,E2 11720.796} C_VEL
LIN {X 0,Y 268.773,Z 217.346,A -85,B 0,C 180,E1 11717.649,E2 11717.649} C_VEL
LIN {X 0,Y 265.125,Z 212.141,A -85,B 0,C 180,E1 11714.971,E2 11714.971} C_VEL
LIN {X 0,Y 262.638,Z 208.797,A -85,B 0,C 180,E1 11712.868,E2 11712.868} C_VEL
LIN {X 0,Y 259.603,Z 204.517,A -85,B 0,C 180,E1 11709.756,E2 11709.756} C_VEL
LIN {X 0,Y 255.818,Z 199.315,A -85,B 0,C 180,E1 11704.034,E2 11704.034} C_VEL
LIN {X 0,Y 254.127,Z 198.122,A -85,B 0,C 180,E1 11697.898,E2 11697.898} C_VEL
LIN {X 0,Y 254.897,Z 198.852,A -85,B 0,C 180,E1 11692.335,E2 11692.335} C_VEL
LIN {X 0,Y 255.588,Z 199.689,A -85,B 0,C 180,E1 11690.543,E2 11690.543} C_VEL
LIN {X 0,Y 259.054,Z 204.735,A -85,B 0,C 180,E1 11685.013,E2 11685.013} C_VEL
LIN {X 0,Y 262.347,Z 209.377,A -85,B 0,C 180,E1 11681.558,E2 11681.558} C_VEL
LIN {X 0,Y 266.141,Z 214.978,A -85,B 0,C 180,E1 11678.396,E2 11678.396} C_VEL
LIN {X 0,Y 270.998,Z 222.353,A -85,B 0,C 180,E1 11675.068,E2 11675.068} C_VEL
LIN {X 0,Y 276.148,Z 230.623,A -85,B 0,C 180,E1 11672.077,E2 11672.077} C_VEL
LIN {X 0,Y 281.792,Z 240.422,A -85,B 0,C 180,E1 11669.214,E2 11669.214} C_VEL
LIN {X 0,Y 287.942,Z 251.959,A -85,B 0,C 180,E1 11666.453,E2 11666.453} C_VEL
LIN {X 0,Y 291.151,Z 258.851,A -85,B 0,C 180,E1 11665.105,E2 11665.105} C_VEL
LIN {X 0,Y 281.27,Z 399.735,A -85,B 0,C 180,E1 11662.001,E2 11662.001} C_VEL
LIN {X 0,Y 278.605,Z 419.57,A -85,B 0,C 180,E1 11661.269,E2 11661.269} C_VEL
LIN {X 0,Y 274.965,Z 438.223,A -85,B 0,C 180,E1 11660.269,E2 11660.269} C_VEL
LIN {X 0,Y 270.076,Z 457.235,A -85,B 0,C 180,E1 11658.882,E2 11658.882} C_VEL
LIN {X 0,Y 264.415,Z 474.973,A -85,B 0,C 180,E1 11657.186,E2 11657.186} C_VEL
LIN {X 0,Y 258.107,Z 491.621,A -85,B 0,C 180,E1 11655.144,E2 11655.144} C_VEL
LIN {X 0,Y 251.3,Z 507.196,A -85,B 0,C 180,E1 11652.714,E2 11652.714} C_VEL
LIN {X 0,Y 243.939,Z 522.134,A -85,B 0,C 180,E1 11649.746,E2 11649.746} C_VEL
LIN {X 0,Y 236.979,Z 534.974,A -85,B 0,C 180,E1 11646.504,E2 11646.504} C_VEL
LIN {X 0,Y 230.358,Z 546.338,A -85,B 0,C 180,E1 11642.856,E2 11642.856} C_VEL
LIN {X 0,Y 223.953,Z 556.787,A -85,B 0,C 180,E1 11638.534,E2 11638.534} C_VEL
LIN {X 0,Y 218.728,Z 565.138,A -85,B 0,C 180,E1 11634.005,E2 11634.005} C_VEL
LIN {X 0,Y 214.506,Z 571.976,A -85,B 0,C 180,E1 11629.042,E2 11629.042} C_VEL
LIN {X 0,Y 211.47,Z 577.207,A -85,B 0,C 180,E1 11623.673,E2 11623.673} C_VEL
LIN {X 0,Y 209.732,Z 580.592,A -85,B 0,C 180,E1 11618.221,E2 11618.221} C_VEL
LIN {X 0,Y 209.016,Z 582.26,A -85,B 0,C 180,E1 11612.74,E2 11612.74} C_VEL
LIN {X 0,Y 208.996,Z 582.297,A -85,B 0,C 180,E1 11607.531,E2 11607.531} C_VEL
LIN {X 0,Y 209.602,Z 580.857,A -85,B 0,C 180,E1 11602.322,E2 11602.322} C_VEL
LIN {X 0,Y 211.102,Z 577.881,A -85,B 0,C 180,E1 11597.136,E2 11597.136} C_VEL
LIN {X 0,Y 213.734,Z 573.265,A -85,B 0,C 180,E1 11592.014,E2 11592.014} C_VEL
LIN {X 0,Y 217.662,Z 566.871,A -85,B 0,C 180,E1 11587.015,E2 11587.015} C_VEL
LIN {X 0,Y 222.912,Z 558.505,A -85,B 0,C 180,E1 11582.192,E2 11582.192} C_VEL
LIN {X 0,Y 229.028,Z 548.619,A -85,B 0,C 180,E1 11577.881,E2 11577.881} C_VEL
LIN {X 0,Y 235.561,Z 537.567,A -85,B 0,C 180,E1 11574.142,E2 11574.142} C_VEL
LIN {X 0,Y 242.389,Z 525.221,A -85,B 0,C 180,E1 11570.851,E2 11570.851} C_VEL
LIN {X 0,Y 249.63,Z 510.91,A -85,B 0,C 180,E1 11567.846,E2 11567.846} C_VEL
LIN {X 0,Y 256.58,Z 495.505,A -85,B 0,C 180,E1 11565.299,E2 11565.299} C_VEL
LIN {X 0,Y 263.111,Z 478.91,A -85,B 0,C 180,E1 11563.143,E2 11563.143} C_VEL
LIN {X 0,Y 268.152,Z 463.927,A -85,B 0,C 180,E1 11561.584,E2 11561.584} C_VEL
LIN {X 0,Y 263.037,Z 467.664,A -85,B 0,C 180,E1 11560.847,E2 11560.847} C_VEL
LIN {X 0,Y 257.361,Z 472.456,A -85,B 0,C 180,E1 11560.16,E2 11560.16} C_VEL
LIN {X 0,Y 251.653,Z 476.095,A -85,B 0,C 180,E1 11559.179,E2 11559.179} C_VEL
LIN {X 0,Y 250.077,Z 476.965,A -85,B 0,C 180,E1 11558.883,E2 11558.883} C_VEL
LIN {X 0,Y 244.825,Z 480.741,A -85,B 0,C 180,E1 11558.075,E2 11558.075} C_VEL
LIN {X 0,Y 240.364,Z 483.009,A -85,B 0,C 180,E1 11557.098,E2 11557.098} C_VEL
LIN {X 0,Y 238.89,Z 483.772,A -85,B 0,C 180,E1 11556.764,E2 11556.764} C_VEL
LIN {X 0,Y 238.604,Z 483.985,A -85,B 0,C 180,E1 11556.716,E2 11556.716} C_VEL
LIN {X 0,Y 233.63,Z 488.304,A -85,B 0,C 180,E1 11556.096,E2 11556.096} C_VEL
LIN {X 0,Y 226.558,Z 494.772,A -85,B 0,C 180,E1 11555.361,E2 11555.361} C_VEL
LIN {X 0,Y 222.885,Z 497.149,A -85,B 0,C 180,E1 11554.675,E2 11554.675} C_VEL
LIN {X 0,Y 221.508,Z 497.647,A -85,B 0,C 180,E1 11554.261,E2 11554.261} C_VEL
LIN {X 0,Y 219.854,Z 498.126,A -85,B 0,C 180,E1 11553.7,E2 11553.7} C_VEL
LIN {X 0,Y 216.186,Z 500.087,A -85,B 0,C 180,E1 11552.761,E2 11552.761} C_VEL
LIN {X 0,Y 214.065,Z 500.447,A -85,B 0,C 180,E1 11551.858,E2 11551.858} C_VEL
LIN {X 0,Y 213.531,Z 500.422,A -85,B 0,C 180,E1 11551.457,E2 11551.457} C_VEL
LIN {X 0,Y 210.179,Z 516.314,A -85,B 0,C 180,E1 11548.097,E2 11548.097} C_VEL
LIN {X 0,Y 207.265,Z 530.235,A -85,B 0,C 180,E1 11544.512,E2 11544.512} C_VEL
LIN {X 0,Y 204.784,Z 542.76,A -85,B 0,C 180,E1 11540.582,E2 11540.582} C_VEL
LIN {X 0,Y 202.849,Z 553.869,A -85,B 0,C 180,E1 11536.318,E2 11536.318} C_VEL
LIN {X 0,Y 201.534,Z 563.548,A -85,B 0,C 180,E1 11531.737,E2 11531.737} C_VEL
LIN {X 0,Y 200.867,Z 571.297,A -85,B 0,C 180,E1 11527.149,E2 11527.149} C_VEL
LIN {X 0,Y 200.713,Z 577.657,A -85,B 0,C 180,E1 11522.285,E2 11522.285} C_VEL
LIN {X 0,Y 201.033,Z 582.323,A -85,B 0,C 180,E1 11517.435,E2 11517.435} C_VEL
LIN {X 0,Y 202.059,Z 585.593,A -85,B 0,C 180,E1 11512.323,E2 11512.323} C_VEL
LIN {X 0,Y 204.323,Z 587.345,A -85,B 0,C 180,E1 11506.865,E2 11506.865} C_VEL
LIN {X 0,Y 208.326,Z 587.3,A -85,B 0,C 180,E1 11501.243,E2 11501.243} C_VEL
LIN {X 0,Y 213.956,Z 585.462,A -85,B 0,C 180,E1 11496.011,E2 11496.011} C_VEL
LIN {X 0,Y 221.734,Z 581.704,A -85,B 0,C 180,E1 11490.857,E2 11490.857} C_VEL
LIN {X 0,Y 231.363,Z 576.062,A -85,B 0,C 180,E1 11486.118,E2 11486.118} C_VEL
LIN {X 0,Y 243.368,Z 568.264,A -85,B 0,C 180,E1 11481.657,E2 11481.657} C_VEL
LIN {X 0,Y 253.276,Z 561.393,A -85,B 0,C 180,E1 11478.757,E2 11478.757} C_VEL
LIN {X 0,Y 238.059,Z 573.469,A -85,B 0,C 180,E1 11474.542,E2 11474.542} C_VEL
LIN {X 0,Y 224.366,Z 585.084,A -85,B 0,C 180,E1 11469.159,E2 11469.159} C_VEL
LIN {X 0,Y 213.961,Z 594.787,A -85,B 0,C 180,E1 11463.146,E2 11463.146} C_VEL
LIN {X 0,Y 206.756,Z 602.441,A -85,B 0,C 180,E1 11456.729,E2 11456.729} C_VEL
LIN {X 0,Y 202.485,Z 607.884,A -85,B 0,C 180,E1 11450.224,E2 11450.224} C_VEL
LIN {X 0,Y 200.674,Z 611.069,A -85,B 0,C 180,E1 11444.133,E2 11444.133} C_VEL
LIN {X 0,Y 200.388,Z 612.487,A -85,B 0,C 180,E1 11440.35,E2 11440.35} C_VEL
LIN {X 0,Y 200.544,Z 614.792,A -85,B 0,C 180,E1 11435.151,E2 11435.151} C_VEL
LIN {X 0,Y 200.753,Z 615.558,A -85,B 0,C 180,E1 11430.858,E2 11430.858} C_VEL
LIN {X 0,Y 200.627,Z 615.17,A -85,B 0,C 180,E1 11426.287,E2 11426.287} C_VEL
LIN {X 0,Y 200.396,Z 613.54,A -85,B 0,C 180,E1 11421.682,E2 11421.682} C_VEL
LIN {X 0,Y 200.649,Z 610.044,A -85,B 0,C 180,E1 11416.163,E2 11416.163} C_VEL
LIN {X 0,Y 202.133,Z 604.525,A -85,B 0,C 180,E1 11410.347,E2 11410.347} C_VEL
LIN {X 0,Y 204.98,Z 597.446,A -85,B 0,C 180,E1 11404.891,E2 11404.891} C_VEL
LIN {X 0,Y 209.09,Z 588.974,A -85,B 0,C 180,E1 11399.863,E2 11399.863} C_VEL
LIN {X 0,Y 214.608,Z 578.563,A -85,B 0,C 180,E1 11395.039,E2 11395.039} C_VEL
LIN {X 0,Y 221.481,Z 565.91,A -85,B 0,C 180,E1 11390.469,E2 11390.469} C_VEL
LIN {X 0,Y 228.69,Z 552.451,A -85,B 0,C 180,E1 11386.655,E2 11386.655} C_VEL
LIN {X 0,Y 236.455,Z 537.159,A -85,B 0,C 180,E1 11383.237,E2 11383.237} C_VEL
LIN {X 0,Y 244.129,Z 520.87,A -85,B 0,C 180,E1 11380.381,E2 11380.381} C_VEL
LIN {X 0,Y 251.322,Z 503.867,A -85,B 0,C 180,E1 11378.03,E2 11378.03} C_VEL
LIN {X 0,Y 257.996,Z 485.968,A -85,B 0,C 180,E1 11376.091,E2 11376.091} C_VEL
LIN {X 0,Y 263.947,Z 467.307,A -85,B 0,C 180,E1 11374.525,E2 11374.525} C_VEL
LIN {X 0,Y 269.103,Z 447.677,A -85,B 0,C 180,E1 11373.284,E2 11373.284} C_VEL
LIN {X 0,Y 273.286,Z 426.939,A -85,B 0,C 180,E1 11372.34,E2 11372.34} C_VEL
LIN {X 0,Y 276.082,Z 405.639,A -85,B 0,C 180,E1 11371.656,E2 11371.656} C_VEL
LIN {X 0,Y 287.571,Z 260.84,A -85,B 0,C 180,E1 11368.251,E2 11368.251} C_VEL
LIN {X 0,Y 281.141,Z 248.293,A -85,B 0,C 180,E1 11365.319,E2 11365.319} C_VEL
LIN {X 0,Y 274.213,Z 236.204,A -85,B 0,C 180,E1 11361.721,E2 11361.721} C_VEL
LIN {X 0,Y 269.016,Z 228.066,A -85,B 0,C 180,E1 11358.584,E2 11358.584} C_VEL
LIN {X 0,Y 265.991,Z 223.454,A -85,B 0,C 180,E1 11356.487,E2 11356.487} C_VEL
LIN {X 0,Y 262.708,Z 218.593,A -85,B 0,C 180,E1 11353.873,E2 11353.873} C_VEL
LIN {X 0,Y 258.419,Z 212.393,A -85,B 0,C 180,E1 11349.577,E2 11349.577} C_VEL
LIN {X 0,Y 254.728,Z 207.204,A -85,B 0,C 180,E1 11343.826,E2 11343.826} C_VEL
LIN {X 0,Y 253.144,Z 206.063,A -85,B 0,C 180,E1 11337.79,E2 11337.79} C_VEL
LIN {X 0,Y 253.935,Z 206.813,A -85,B 0,C 180,E1 11332.306,E2 11332.306} C_VEL
LIN {X 0,Y 254.617,Z 207.785,A -85,B 0,C 180,E1 11330.506,E2 11330.506} C_VEL
LIN {X 0,Y 257.819,Z 212.605,A -85,B 0,C 180,E1 11325.284,E2 11325.284} C_VEL
LIN {X 0,Y 260.81,Z 216.953,A -85,B 0,C 180,E1 11322.024,E2 11322.024} C_VEL
LIN {X 0,Y 264.426,Z 222.476,A -85,B 0,C 180,E1 11318.889,E2 11318.889} C_VEL
LIN {X 0,Y 268.91,Z 229.529,A -85,B 0,C 180,E1 11315.682,E2 11315.682} C_VEL
LIN {X 0,Y 273.97,Z 237.92,A -85,B 0,C 180,E1 11312.623,E2 11312.623} C_VEL
LIN {X 0,Y 279.712,Z 248.23,A -85,B 0,C 180,E1 11309.615,E2 11309.615} C_VEL
LIN {X 0,Y 286.221,Z 261.112,A -85,B 0,C 180,E1 11306.607,E2 11306.607} C_VEL
LIN {X 0,Y 286.694,Z 262.565,A -85,B 0,C 180,E1 11306.381,E2 11306.381} C_VEL
LIN {X 0,Y 276.674,Z 400.044,A -85,B 0,C 180,E1 11303.345,E2 11303.345} C_VEL
LIN {X 0,Y 273.923,Z 419.872,A -85,B 0,C 180,E1 11302.614,E2 11302.614} C_VEL
LIN {X 0,Y 270.125,Z 438.7,A -85,B 0,C 180,E1 11301.606,E2 11301.606} C_VEL
LIN {X 0,Y 265.235,Z 457.173,A -85,B 0,C 180,E1 11300.264,E2 11300.264} C_VEL
LIN {X 0,Y 259.377,Z 475.008,A -85,B 0,C 180,E1 11298.568,E2 11298.568} C_VEL
LIN {X 0,Y 252.844,Z 491.723,A -85,B 0,C 180,E1 11296.521,E2 11296.521} C_VEL
LIN {X 0,Y 245.495,Z 507.941,A -85,B 0,C 180,E1 11293.978,E2 11293.978} C_VEL
LIN {X 0,Y 238.356,Z 521.913,A -85,B 0,C 180,E1 11291.19,E2 11291.19} C_VEL
LIN {X 0,Y 231.051,Z 534.87,A -85,B 0,C 180,E1 11287.913,E2 11287.913} C_VEL
LIN {X 0,Y 224.071,Z 546.344,A -85,B 0,C 180,E1 11284.209,E2 11284.209} C_VEL
LIN {X 0,Y 217.622,Z 556.372,A -85,B 0,C 180,E1 11280.051,E2 11280.051} C_VEL
LIN {X 0,Y 211.966,Z 564.928,A -85,B 0,C 180,E1 11275.418,E2 11275.418} C_VEL
LIN {X 0,Y 207.546,Z 571.63,A -85,B 0,C 180,E1 11270.588,E2 11270.588} C_VEL
LIN {X 0,Y 204.196,Z 576.954,A -85,B 0,C 180,E1 11265.283,E2 11265.283} C_VEL
LIN {X 0,Y 202.093,Z 580.657,A -85,B 0,C 180,E1 11259.682,E2 11259.682} C_VEL
LIN {X 0,Y 201.149,Z 582.595,A -85,B 0,C 180,E1 11254.274,E2 11254.274} C_VEL
LIN {X 0,Y 200.971,Z 583.045,A -85,B 0,C 180,E1 11248.858,E2 11248.858} C_VEL
LIN {X 0,Y 201.427,Z 582.027,A -85,B 0,C 180,E1 11243.442,E2 11243.442} C_VEL
LIN {X 0,Y 202.768,Z 579.494,A -85,B 0,C 180,E1 11238.046,E2 11238.046} C_VEL
LIN {X 0,Y 205.26,Z 575.333,A -85,B 0,C 180,E1 11232.701,E2 11232.701} C_VEL
LIN {X 0,Y 209.333,Z 569.014,A -85,B 0,C 180,E1 11227.199,E2 11227.199} C_VEL
LIN {X 0,Y 214.563,Z 561.133,A -85,B 0,C 180,E1 11222.223,E2 11222.223} C_VEL
LIN {X 0,Y 220.437,Z 552.209,A -85,B 0,C 180,E1 11217.946,E2 11217.946} C_VEL
LIN {X 0,Y 227.352,Z 541.228,A -85,B 0,C 180,E1 11213.89,E2 11213.89} C_VEL
LIN {X 0,Y 234.747,Z 528.663,A -85,B 0,C 180,E1 11210.289,E2 11210.289} C_VEL
LIN {X 0,Y 242.142,Z 514.943,A -85,B 0,C 180,E1 11207.213,E2 11207.213} C_VEL
LIN {X 0,Y 249.56,Z 499.551,A -85,B 0,C 180,E1 11204.506,E2 11204.506} C_VEL
LIN {X 0,Y 256.54,Z 482.942,A -85,B 0,C 180,E1 11202.222,E2 11202.222} C_VEL
LIN {X 0,Y 258.567,Z 477.358,A -85,B 0,C 180,E1 11201.558,E2 11201.558} C_VEL
LIN {X 0,Y 252.058,Z 481.483,A -85,B 0,C 180,E1 11200.584,E2 11200.584} C_VEL
LIN {X 0,Y 249.603,Z 482.888,A -85,B 0,C 180,E1 11200.161,E2 11200.161} C_VEL
LIN {X 0,Y 243.451,Z 486.93,A -85,B 0,C 180,E1 11199.234,E2 11199.234} C_VEL
LIN {X 0,Y 237.203,Z 490.068,A -85,B 0,C 180,E1 11197.976,E2 11197.976} C_VEL
LIN {X 0,Y 231.647,Z 493.199,A -85,B 0,C 180,E1 11196.868,E2 11196.868} C_VEL
LIN {X 0,Y 228.273,Z 494.422,A -85,B 0,C 180,E1 11195.94,E2 11195.94} C_VEL
LIN {X 0,Y 223.606,Z 496.95,A -85,B 0,C 180,E1 11194.915,E2 11194.915} C_VEL
LIN {X 0,Y 221.508,Z 497.647,A -85,B 0,C 180,E1 11194.261,E2 11194.261} C_VEL
LIN {X 0,Y 217.426,Z 499.23,A -85,B 0,C 180,E1 11193.005,E2 11193.005} C_VEL
LIN {X 0,Y 212.301,Z 502.575,A -85,B 0,C 180,E1 11191.774,E2 11191.774} C_VEL
LIN {X 0,Y 206.355,Z 508.522,A -85,B 0,C 180,E1 11190.325,E2 11190.325} C_VEL
LIN {X 0,Y 203.106,Z 514.015,A -85,B 0,C 180,E1 11189.118,E2 11189.118} C_VEL
LIN {X 0,Y 202.338,Z 516.493,A -85,B 0,C 180,E1 11188.545,E2 11188.545} C_VEL
LIN {X 0,Y 199.186,Z 531.153,A -85,B 0,C 180,E1 11184.623,E2 11184.623} C_VEL
LIN {X 0,Y 196.517,Z 544.404,A -85,B 0,C 180,E1 11180.242,E2 11180.242} C_VEL
LIN {X 0,Y 194.524,Z 556.002,A -85,B 0,C 180,E1 11175.503,E2 11175.503} C_VEL
